	ERROR
		IF ERRNO = ERR_FILEOPEN THEN
			TPWrite "ERROR: Cannot open config.txt or log file";
		ELSE
			TPWrite "ERROR in TestGantryFloorCoordinates: " + NumToStr(ERRNO, 0);
		ENDIF
		Close configfile;
		Close debug_logfile;
		STOP;
	ENDPROC

	! ========================================
	! Test Gantry with Multiple R-axis Rotations
	! ========================================
	! Version: v1.8.7
	! Date: 2026-01-05
	! Purpose: Test Robot1 and Robot2 TCP positions at various R-axis angles
	! Features:
	!   - Config-based angle configuration (NUM_R_ANGLES, R_ANGLE_1~10)
	!   - Robot1 and Robot2 Floor TCP coordinate measurement
	!   - Automatic gantry position logging
	! Changes in v1.8.7:
	!   - Reduced header writes and summarized R_ANGLES for 41617 stability
	!   - Increased per-angle WaitTime to 0.2 for I/O stability
	! Changes in v1.8.5:
	!   - Log gantry Floor values using Floor conversion (X+9500, Y/Z inverted)
	! Changes in v1.8.4:
	!   - Chunked file logging with WaitTime 0.1 to reduce 41617
	! Changes in v1.8.1:
	!   - BUGFIX: Added UpdateRobot2BaseDynamicWobj() call (Line 1918)
	!   - Fixed Robot2 Floor TCP reporting [0,0,0]
	! Changes in v1.8.0:
	!   - Config-based R-axis angle reading from config.txt
	!   - Replaces hardcoded angles with NUM_R_ANGLES and R_ANGLE_1~10
	!   - Enhanced logging with gantry position details
	! Initial position: Robot1 and Robot2 at HOME
	! Gantry position: X=0, Y=0, Z=0 (fixed), R varies according to config
	! Output: /HOME/gantry_rotation_test.txt
	PROC TestGantryRotation()
		VAR jointtarget home_pos;
		VAR jointtarget test_pos;
		VAR robtarget rob1_floor;
		VAR robtarget rob2_floor;
		VAR iodev logfile;
		VAR iodev configfile;
		VAR num test_x;
		VAR num test_y;
		VAR num test_z;
		VAR num r_angles{10};
		VAR num num_r_angles;
		VAR num i;
		VAR string r_str;
		VAR string line;
		VAR string value_str;
		VAR string r_list;
		VAR string csv_line;
		VAR bool found_value;

		! Initialize
		test_x := 0;  ! Fixed at 0 for R-axis rotation test
		test_y := 0;
		test_z := 0;
		num_r_angles := 0;

		! Read config.txt for R angles
		TPWrite "Reading config.txt for R angles...";
		Open "HOME:/config.txt", configfile \Read;

		! Read NUM_R_ANGLES
		WHILE num_r_angles = 0 DO
			line := ReadStr(configfile \RemoveCR);
			IF StrFind(line, 1, "NUM_R_ANGLES=") = 1 THEN
				IF StrLen(line) >= 14 THEN
					value_str := StrPart(line, 14, StrLen(line) - 13);
					found_value := StrToVal(value_str, num_r_angles);
					TPWrite "NUM_R_ANGLES=" + NumToStr(num_r_angles, 0);
				ENDIF
			ENDIF
		ENDWHILE

		! Read R_ANGLE_1 to R_ANGLE_10
		FOR i FROM 1 TO num_r_angles DO
			WHILE TRUE DO
				line := ReadStr(configfile);
				IF StrFind(line, 1, "R_ANGLE_" + NumToStr(i,0) + "=") = 1 THEN
					value_str := StrPart(line, StrLen("R_ANGLE_" + NumToStr(i,0) + "=") + 1, StrLen(line) - StrLen("R_ANGLE_" + NumToStr(i,0) + "="));
					found_value := StrToVal(value_str, r_angles{i});
					TPWrite "R_ANGLE_" + NumToStr(i,0) + "=" + NumToStr(r_angles{i}, 1);
					GOTO next_angle;
				ENDIF
			ENDWHILE
			next_angle:
		ENDFOR

		Close configfile;

		! Build R angle list for header logging
		r_list := "";
		FOR i FROM 1 TO num_r_angles DO
			IF i = 1 THEN
				r_list := NumToStr(r_angles{i}, 1);
			ELSE
				r_list := r_list + "," + NumToStr(r_angles{i}, 1);
			ENDIF
		ENDFOR

		TPWrite "========================================";
		TPWrite "Starting Multiple R-axis Rotation Test";
		TPWrite "========================================";

		! Verify initial position
		TPWrite "Verifying robots at HOME position...";
		home_pos := CJointT();
		IF Abs(home_pos.extax.eax_a) > 10 OR Abs(home_pos.extax.eax_b) > 10 OR Abs(home_pos.extax.eax_c) > 10 OR Abs(home_pos.extax.eax_d) > 2 THEN
			TPWrite "WARNING: Gantry not at HOME!";
			TPWrite "Current: [" + NumToStr(home_pos.extax.eax_a,0) + ", " + NumToStr(home_pos.extax.eax_b,0) + ", " + NumToStr(home_pos.extax.eax_c,0) + ", " + NumToStr(home_pos.extax.eax_d,1) + "]";
			TPWrite "Please run SetRobot1InitialPosition first";
			RETURN;
		ENDIF

		! Open log file (reduced header writes)
		Open "HOME:/gantry_rotation_test.txt", logfile \Write;
		Write logfile, "Gantry R-axis Rotation Test (" + TASK1_VERSION + ")";
		Write logfile, "Date=" + CDate() + ", Time=" + CTime();
		Write logfile, "Gantry Phys=[" + NumToStr(test_x,0) + "," + NumToStr(test_y,0) + "," + NumToStr(test_z,0)
		              + "], Floor=[" + NumToStr(test_x + 9500,0) + "," + NumToStr(5300 - test_y,0) + "," + NumToStr(2100 - test_z,0) + "]";
		Write logfile, "R_ANGLES=" + r_list;
		Write logfile, "Floor: X+=right, Y+=up, Z+=up, R0:Y-axis, R1 Y+, R2 Y-";
		Write logfile, "R_DEG,GX,GY,GZ,R1X,R1Y,R1Z,R2X,R2Y,R2Z";
		WaitTime 0.3;

		! Test each R angle
		FOR i FROM 1 TO num_r_angles DO
			r_str := NumToStr(r_angles{i}, 1);
			TPWrite "----------------------------------------";
			TPWrite "Test " + NumToStr(i,0) + "/" + NumToStr(num_r_angles,0) + ": R = " + r_str + " degrees";
			TPWrite "----------------------------------------";

			! Move gantry to test position with current R angle
			test_pos := CJointT();
			test_pos.extax.eax_a := test_x;
			test_pos.extax.eax_b := test_y;
			test_pos.extax.eax_c := test_z;
			test_pos.extax.eax_d := r_angles{i};
			test_pos.extax.eax_f := test_x;  ! X2 = X1 (synchronized)
			MoveAbsJ test_pos, v100, fine, tool0;
			WaitTime 0.5;

			! Measure Floor positions
			UpdateRobot1FloorPosition;
			UpdateRobot2BaseDynamicWobj;  ! Update Robot2 base coordinate for TASK2
			! Note: robot2_floor_pos_t1 is updated by UpdateRobot2BaseDynamicWobj
			rob1_floor := robot1_floor_pos_t1;
			rob2_floor := robot2_floor_pos_t1;  ! Updated by TASK2

			! Write results to file (1-line CSV)
			csv_line := NumToStr(r_angles{i}, 1) + ","
			          + NumToStr(test_pos.extax.eax_a,0) + "," + NumToStr(test_pos.extax.eax_b,0) + "," + NumToStr(test_pos.extax.eax_c,0) + ","
			          + NumToStr(rob1_floor.trans.x, 2) + "," + NumToStr(rob1_floor.trans.y, 2) + "," + NumToStr(rob1_floor.trans.z, 2) + ","
			          + NumToStr(rob2_floor.trans.x, 2) + "," + NumToStr(rob2_floor.trans.y, 2) + "," + NumToStr(rob2_floor.trans.z, 2);
			Write logfile, csv_line;
			WaitTime 0.2; ! Keep this WaitTime for I/O stability
			! Display on teach pendant
			TPWrite "Robot1 Floor: [" + NumToStr(rob1_floor.trans.x,1) + ", " + NumToStr(rob1_floor.trans.y,1) + ", " + NumToStr(rob1_floor.trans.z,1) + "]";
			TPWrite "Robot2 Floor: [" + NumToStr(rob2_floor.trans.x,1) + ", " + NumToStr(rob2_floor.trans.y,1) + ", " + NumToStr(rob2_floor.trans.z,1) + "]";
		ENDFOR

		! Return to HOME
		TPWrite "Returning to HOME...";
		MoveAbsJ home_pos, v100, fine, tool0;

		Write logfile, "========================================";
		Write logfile, "Test completed - Returned to HOME";
		Write logfile, "========================================";
		Close logfile;

		TPWrite "========================================";
		TPWrite "R-axis Rotation Test Complete!";
		TPWrite "Results saved to gantry_rotation_test.txt";
		TPWrite "========================================";

	ERROR
		IF ERRNO = ERR_FILEOPEN THEN
			TPWrite "ERROR: Cannot open log file";
		ELSE
			TPWrite "ERROR in TestGantryRotation: " + NumToStr(ERRNO, 0);
		ENDIF
		Close logfile;
		STOP;
	ENDPROC

	! ========================================
	! Mode 2 - Gantry + TCP Offset Verification
	! ========================================
		! Version: v1.8.50
		! Date: 2026-01-08
		! Purpose: Verify TCP tracking with offsets while gantry moves in X/Y/Z/R
		! Config (config.txt):
		!   TEST_MODE=2
		!   TCP_OFFSET_R1_X/Y/Z (fallback: TCP_OFFSET_X/Y/Z)
		!   NUM_POS, POS_1_X/Y/Z/R ...
	! Output: /HOME/gantry_mode2_test.txt
		! Changes in v1.8.50:
		!   - Use hardcoded Mode2 defaults (config.txt ignored).
		! Changes in v1.8.49:
		!   - Remove CONTINUE usage in Mode2 parse loop for RAPID compatibility.
		! Changes in v1.8.48:
		!   - Rework Mode2 config parsing: single-pass ReadStr loop with guards.
		! Changes in v1.8.47:
		!   - TEMP: Bypass config.txt parsing and use default Mode2 offsets/positions.
		! Changes in v1.8.46:
		!   - Use ReadStr \RemoveCR in Mode2 parsing loops to avoid blocking on CRLF files.
		! Changes in v1.8.14:
		!   - Align gantry axis range checks with MOC.cfg (M1/M2/M3/M4 limits)

! ========================================
! Mode 2 - Gantry + TCP Offset Verification (v1.8.51)
! ========================================
! Version: v1.8.51
! Date: 2026-01-08
! Purpose: Verify TCP tracking with offsets using PERS variables
! No config.txt parsing - all settings from PERS variables
! Output: /HOME/gantry_mode2_test.txt
PROC TestGantryMode2()
	VAR jointtarget home_pos;
	VAR jointtarget test_pos;
	VAR robtarget offset_tcp;
	VAR robtarget rob1_floor;
	VAR robtarget rob2_floor;
	VAR iodev logfile;
	VAR num tcp_offset_x;
	VAR num tcp_offset_y;
	VAR num tcp_offset_z;
	VAR num num_pos;
	VAR num pos_x{10};
	VAR num pos_y{10};
	VAR num pos_z{10};
	VAR num pos_r{10};
	VAR num i;
	VAR string csv_line;
	VAR num floor_x;
	VAR num floor_y;
	VAR num floor_z;
	VAR num floor_r;
	VAR num phys_x;
	VAR num phys_y;
	VAR num phys_z;
	VAR num phys_r;
	VAR bool abort_test;
	VAR string mode2_log;
	VAR string tp_log;
	VAR iodev tp_logfile;
	VAR jointtarget current_gantry;
	VAR robjoint robot1_offset_joints;
	VAR num wait_count;

	abort_test := FALSE;
	mode2_log := "HOME:/gantry_mode2_test.txt";
	tp_log := "HOME:/tp_messages.txt";

	! v1.8.57: Reset sync flags at start (TASK2 must wait)
	mode2_config_ready := FALSE;
	mode2_r2_initial_offset_done := FALSE;

	Open mode2_log, logfile \Write;
	Open tp_log, tp_logfile \Write;
	Write tp_logfile, "TP Log (" + TASK1_VERSION + ") Date=" + CDate() + " Time=" + CTime();
	Write tp_logfile, "========================================";
	Write logfile, "Mode2 Test (" + TASK1_VERSION + ") Date=" + CDate() + " Time=" + CTime();
	Write logfile, "Enter TestGantryMode2";
	TPWrite "Mode2: Loading config from PERS variables";
	Write tp_logfile, "Mode2: Loading config from PERS variables";

	! DEBUG: Log ConfigModule PERS values BEFORE copy
	Write tp_logfile, "DEBUG: ConfigModule R2 BEFORE copy:";
	Write tp_logfile, "  MODE2_TCP_OFFSET_R2_X=" + NumToStr(MODE2_TCP_OFFSET_R2_X, 1);
	Write tp_logfile, "  MODE2_TCP_OFFSET_R2_Y=" + NumToStr(MODE2_TCP_OFFSET_R2_Y, 1);
	Write tp_logfile, "  MODE2_TCP_OFFSET_R2_Z=" + NumToStr(MODE2_TCP_OFFSET_R2_Z, 1);
	Write tp_logfile, "DEBUG: mode2_r2_offset BEFORE copy:";
	Write tp_logfile, "  mode2_r2_offset_y=" + NumToStr(mode2_r2_offset_y, 1);

	! Read configuration from PERS variables (no file I/O)
	tcp_offset_x := MODE2_TCP_OFFSET_R1_X;
	tcp_offset_y := MODE2_TCP_OFFSET_R1_Y;
	tcp_offset_z := MODE2_TCP_OFFSET_R1_Z;

	! Sync Robot2 offsets from ConfigModule (for TASK2)
	mode2_r2_offset_x := MODE2_TCP_OFFSET_R2_X;
	mode2_r2_offset_y := MODE2_TCP_OFFSET_R2_Y;
	mode2_r2_offset_z := MODE2_TCP_OFFSET_R2_Z;

	! v1.8.57: Set sync flag (TASK2 can now read values)
	mode2_config_ready := TRUE;
	Write tp_logfile, "SYNC: mode2_config_ready=TRUE (TASK2 can proceed)";

	! DEBUG: Log values AFTER copy
	Write tp_logfile, "DEBUG: mode2_r2_offset AFTER copy:";
	Write tp_logfile, "  mode2_r2_offset_y=" + NumToStr(mode2_r2_offset_y, 1);

	! Log Robot2 offsets
	Write logfile, "R2_OFFSET=" + NumToStr(mode2_r2_offset_x, 1) + ","
	              + NumToStr(mode2_r2_offset_y, 1) + ","
	              + NumToStr(mode2_r2_offset_z, 1);

	! Read test positions
	num_pos := MODE2_NUM_POS;
	FOR i FROM 1 TO 10 DO
		pos_x{i} := MODE2_POS_X{i};
		pos_y{i} := MODE2_POS_Y{i};
		pos_z{i} := MODE2_POS_Z{i};
		pos_r{i} := MODE2_POS_R{i};
	ENDFOR

	Write logfile, "Config loaded from PERS - NUM_POS=" + NumToStr(num_pos, 0);
	Write logfile, "TCP_OFFSET_R1=" + NumToStr(tcp_offset_x,1) + ","
	              + NumToStr(tcp_offset_y,1) + ","
	              + NumToStr(tcp_offset_z,1);
	Write logfile, "X,Y,Z,R,R1X,R1Y,R1Z,R2X,R2Y,R2Z";
	TPWrite "Mode2: Config loaded, NUM_POS=" + NumToStr(num_pos, 0);
	Write tp_logfile, "Mode2: Config loaded, NUM_POS=" + NumToStr(num_pos, 0);
	WaitTime 0.3;

	! Move Robot1 to offset in WobjGantry
	UpdateGantryWobj;
	home_pos := CJointT();
	offset_tcp := [[tcp_offset_x, tcp_offset_y, 1000 + tcp_offset_z], [0.5, -0.5, 0.5, 0.5], [0, 0, 0, 0], home_pos.extax];
	MoveJ offset_tcp, v100, fine, tool0\WObj:=WobjGantry;
	TPWrite "Mode2: Robot1 at offset TCP";
	Write tp_logfile, "Mode2: Robot1 at offset TCP";

	! Save Robot1 joint angles for use in loop (fixed joints = fixed TCP direction)
	current_gantry := CJointT();
	robot1_offset_joints := current_gantry.robax;
	Write tp_logfile, "Robot1 offset joints: saved";

	! v1.8.67: Wait for Robot2 initial offset before moving gantry
	TPWrite "Mode2: Waiting for Robot2 initial offset...";
	Write tp_logfile, "SYNC: Waiting for Robot2 initial offset...";
	wait_count := 0;
	WHILE NOT mode2_r2_initial_offset_done AND wait_count < 100 DO
		WaitTime 0.1;
		wait_count := wait_count + 1;
	ENDWHILE
	IF mode2_r2_initial_offset_done THEN
		Write tp_logfile, "SYNC: Robot2 initial offset done (waited " + NumToStr(wait_count, 0) + " cycles)";
		TPWrite "Mode2: Robot2 initial offset done";
	ELSE
		Write tp_logfile, "WARNING: Robot2 initial offset timeout!";
		TPWrite "Mode2: WARNING - Robot2 offset timeout!";
	ENDIF

	! Test each position
	FOR i FROM 1 TO num_pos DO
		! Calculate Floor coordinates (COMPLEX_POS format)
		floor_x := 9500 + pos_x{i};
		floor_y := 5300 + pos_y{i};
		floor_z := 2100 + pos_z{i};
		floor_r := pos_r{i};

		! Convert to physical gantry coordinates
		phys_x := floor_x - 9500;
		phys_y := 5300 - floor_y;
		phys_z := 2100 - floor_z;
		phys_r := 0 - floor_r;

		! Check gantry axis limits (MOC.cfg)
		! M1 [-9.51, 12.31], M2 [-0.05, 5.35], M3 [-0.05, 1.05], M4 [-100, 100] deg
		IF phys_x < -9510 OR phys_x > 12310 OR phys_y < -50 OR phys_y > 5350 OR phys_z < -50 OR phys_z > 1050 OR phys_r < -100 OR phys_r > 100 THEN
			Write logfile, "OUT_OF_RANGE idx=" + NumToStr(i,0)
			              + " floor=[" + NumToStr(floor_x,0) + "," + NumToStr(floor_y,0) + "," + NumToStr(floor_z,0) + "," + NumToStr(floor_r,1) + "]"
			              + " phys=[" + NumToStr(phys_x,0) + "," + NumToStr(phys_y,0) + "," + NumToStr(phys_z,0) + "," + NumToStr(phys_r,1) + "]";
			TPWrite "Mode2: Position " + NumToStr(i,0) + " out of range!";
			abort_test := TRUE;
			GOTO mode2_cleanup;
		ENDIF

		! Move gantry to test position (Robot1 joints fixed to offset position)
		test_pos := CJointT();
		test_pos.robax := robot1_offset_joints;  ! Keep Robot1 at offset position
		test_pos.extax.eax_a := phys_x;
		test_pos.extax.eax_b := phys_y;
		test_pos.extax.eax_c := phys_z;
		test_pos.extax.eax_d := phys_r;
		test_pos.extax.eax_f := test_pos.extax.eax_a;
		MoveAbsJ test_pos, v100, fine, tool0;
		TPWrite "Mode2: Gantry moved to position " + NumToStr(i,0) + "/" + NumToStr(num_pos,0);
		Write tp_logfile, "Mode2: Gantry moved to position " + NumToStr(i,0) + "/" + NumToStr(num_pos,0);

		! Update WobjGantry for new gantry position and rotation
		UpdateGantryWobj;

		! Read current gantry position AFTER move (fix for eax_e mismatch)
		current_gantry := CJointT();
		Write tp_logfile, "WobjGantry updated: [" + NumToStr(current_gantry.extax.eax_a,0) + ", "
		                  + NumToStr(current_gantry.extax.eax_b,0) + ", "
		                  + NumToStr(current_gantry.extax.eax_c,0) + ", R="
		                  + NumToStr(current_gantry.extax.eax_d,1) + "]";
		Write tp_logfile, "current_gantry.extax: [" + NumToStr(current_gantry.extax.eax_a,1) + ", "
		                  + NumToStr(current_gantry.extax.eax_b,1) + ", "
		                  + NumToStr(current_gantry.extax.eax_c,1) + ", "
		                  + NumToStr(current_gantry.extax.eax_d,1) + ", "
		                  + NumToStr(current_gantry.extax.eax_e,1) + ", "
		                  + NumToStr(current_gantry.extax.eax_f,1) + "]";

		! Robot1 already at offset position (joints fixed in MoveAbsJ)
		Write tp_logfile, "Robot1 maintaining offset joints (pos " + NumToStr(i,0) + ")";

		! v1.8.63: Trigger Robot2 to reposition at current R angle
		mode2_r2_reposition_done := FALSE;
		mode2_r2_reposition_trigger := TRUE;
		Write tp_logfile, "SYNC: Waiting for Robot2 reposition...";
		wait_count := 0;
		WHILE NOT mode2_r2_reposition_done AND wait_count < 100 DO
			WaitTime 0.1;
			wait_count := wait_count + 1;
		ENDWHILE
		mode2_r2_reposition_trigger := FALSE;
		IF mode2_r2_reposition_done THEN
			Write tp_logfile, "SYNC: Robot2 repositioned (waited " + NumToStr(wait_count, 0) + " cycles)";
		ELSE
			Write tp_logfile, "SYNC: WARNING - Robot2 reposition timeout!";
		ENDIF
		WaitTime 0.3;

		! Measure Robot1 and Robot2 TCP positions
		UpdateRobot1FloorPosition;
		UpdateRobot2BaseDynamicWobj;
		rob1_floor := robot1_floor_pos_t1;
		rob2_floor := robot2_floor_pos_t1;

		! v1.8.60 DEBUG: Detailed position analysis
		Write tp_logfile, "========== v1.8.60 DETAILED DEBUG ==========";
		Write tp_logfile, "--- Gantry Position ---";
		Write tp_logfile, "  Gantry Floor: [" + NumToStr(floor_x, 0) + ", " + NumToStr(floor_y, 0) + ", " + NumToStr(floor_z, 0) + "]";
		Write tp_logfile, "  Gantry Local (extax): [" + NumToStr(phys_x, 0) + ", " + NumToStr(phys_y, 0) + ", " + NumToStr(phys_z, 0) + ", R=" + NumToStr(phys_r, 1) + "]";
		Write tp_logfile, "  R-center Floor: [" + NumToStr(floor_x, 0) + ", " + NumToStr(floor_y, 0) + ", " + NumToStr(floor_z, 0) + "]";
		Write tp_logfile, "";
		Write tp_logfile, "--- Robot1 (wobj0 at R-center, gantry-configured) ---";
		Write tp_logfile, "  Robot1 Base Floor = R-center: [" + NumToStr(floor_x, 0) + ", " + NumToStr(floor_y, 0) + ", " + NumToStr(floor_z, 0) + "]";
		Write tp_logfile, "  Robot1 offset_tcp in WobjGantry: [" + NumToStr(tcp_offset_x, 1) + ", " + NumToStr(tcp_offset_y, 1) + ", " + NumToStr(1000 + tcp_offset_z, 1) + "]";
		Write tp_logfile, "  Robot1 TCP Floor (measured): [" + NumToStr(rob1_floor.trans.x, 2) + ", " + NumToStr(rob1_floor.trans.y, 2) + ", " + NumToStr(rob1_floor.trans.z, 2) + "]";
		Write tp_logfile, "  Robot1 TCP offset from R-center: [" + NumToStr(rob1_floor.trans.x - floor_x, 2) + ", " + NumToStr(rob1_floor.trans.y - floor_y, 2) + ", " + NumToStr(rob1_floor.trans.z - floor_z, 2) + "]";
		Write tp_logfile, "";
		Write tp_logfile, "--- Robot2 (wobj0 at Robot2 base, NOT gantry-configured) ---";
		Write tp_logfile, "  Robot2 Base Floor: [" + NumToStr(debug_r2_base_floor_x, 2) + ", " + NumToStr(rob2_floor.trans.y - (debug_r2_wobj0_y * Cos(current_gantry.extax.eax_d)), 2) + "]";
		Write tp_logfile, "  Robot2 offset_tcp in WobjGantry_Rob2: [0, " + NumToStr(488 + mode2_r2_offset_y, 1) + ", -1000]";
		Write tp_logfile, "  Robot2 wobj0 (TCP from base): [" + NumToStr(debug_r2_wobj0_x, 2) + ", " + NumToStr(debug_r2_wobj0_y, 2) + "]";
		Write tp_logfile, "  Robot2 TCP Floor (measured): [" + NumToStr(rob2_floor.trans.x, 2) + ", " + NumToStr(rob2_floor.trans.y, 2) + ", " + NumToStr(rob2_floor.trans.z, 2) + "]";
		Write tp_logfile, "  Robot2 TCP offset from R-center: [" + NumToStr(rob2_floor.trans.x - floor_x, 2) + ", " + NumToStr(rob2_floor.trans.y - floor_y, 2) + ", " + NumToStr(rob2_floor.trans.z - floor_z, 2) + "]";
		Write tp_logfile, "";
		Write tp_logfile, "--- Comparison ---";
		Write tp_logfile, "  3D Distance: " + NumToStr(Sqrt(Pow(rob1_floor.trans.x - rob2_floor.trans.x, 2) + Pow(rob1_floor.trans.y - rob2_floor.trans.y, 2) + Pow(rob1_floor.trans.z - rob2_floor.trans.z, 2)), 2) + " mm";
		Write tp_logfile, "  Expected (at R=0): 200.00 mm";
		Write tp_logfile, "=========================================";

		! v1.8.61 DEBUG: Log X coordinate analysis
		Write tp_logfile, "DEBUG X Analysis:";
		Write tp_logfile, "  Gantry X (R-center): " + NumToStr(phys_x + 9500, 1);
		Write tp_logfile, "  R angle (extax.eax_d): " + NumToStr(current_gantry.extax.eax_d, 1);
		Write tp_logfile, "  sin(R): " + NumToStr(Sin(current_gantry.extax.eax_d), 4);
		Write tp_logfile, "  Robot2 wobj0: [" + NumToStr(debug_r2_wobj0_x, 1) + ", " + NumToStr(debug_r2_wobj0_y, 1) + "]";
		Write tp_logfile, "  Robot2 base_floor_x: " + NumToStr(debug_r2_base_floor_x, 1);
		Write tp_logfile, "  Robot2 floor_x_offset: " + NumToStr(debug_r2_floor_x_offset, 1);
		Write tp_logfile, "  Robot2 X = base + offset: " + NumToStr(debug_r2_base_floor_x, 1) + " + " + NumToStr(debug_r2_floor_x_offset, 1) + " = " + NumToStr(rob2_floor.trans.x, 1);
		Write tp_logfile, "  Robot1 X: " + NumToStr(rob1_floor.trans.x, 2) + " (offset from gantry: " + NumToStr(rob1_floor.trans.x - (phys_x + 9500), 2) + ")";
		Write tp_logfile, "  Robot2 X: " + NumToStr(rob2_floor.trans.x, 2) + " (offset from gantry: " + NumToStr(rob2_floor.trans.x - (phys_x + 9500), 2) + ")";
		Write tp_logfile, "  Expected R2 X offset: +" + NumToStr(100 * Sin(current_gantry.extax.eax_d), 2);
		Write tp_logfile, "  Delta X (R1-R2): " + NumToStr(rob1_floor.trans.x - rob2_floor.trans.x, 2);

		! v1.8.61 DEBUG: Log Y coordinate analysis
		Write tp_logfile, "DEBUG Y Analysis:";
		Write tp_logfile, "  Gantry Y (R-center): " + NumToStr(5300 - phys_y, 1);
		Write tp_logfile, "  cos(R): " + NumToStr(Cos(current_gantry.extax.eax_d), 4);
		Write tp_logfile, "  Robot2 base_floor_y: " + NumToStr(debug_r2_base_floor_y, 1);
		Write tp_logfile, "  Robot2 floor_y_offset: " + NumToStr(debug_r2_floor_y_offset, 1);
		Write tp_logfile, "  Robot2 Y = base + offset: " + NumToStr(debug_r2_base_floor_y, 1) + " + " + NumToStr(debug_r2_floor_y_offset, 1) + " = " + NumToStr(rob2_floor.trans.y, 1);
		Write tp_logfile, "  Robot1 Y: " + NumToStr(rob1_floor.trans.y, 2) + " (offset from gantry: " + NumToStr(rob1_floor.trans.y - (5300 - phys_y), 2) + ")";
		Write tp_logfile, "  Robot2 Y: " + NumToStr(rob2_floor.trans.y, 2) + " (offset from gantry: " + NumToStr(rob2_floor.trans.y - (5300 - phys_y), 2) + ")";
		Write tp_logfile, "  Expected R1 Y offset: +" + NumToStr(100 * Cos(current_gantry.extax.eax_d), 2);
		Write tp_logfile, "  Expected R2 Y offset: -" + NumToStr(100 * Cos(current_gantry.extax.eax_d), 2);
		Write tp_logfile, "  Delta Y (R1-R2): " + NumToStr(rob1_floor.trans.y - rob2_floor.trans.y, 2);
		Write tp_logfile, "  Expected Delta Y: " + NumToStr(200 * Cos(current_gantry.extax.eax_d), 2);

		Write tp_logfile, "Robot1 Floor: [" + NumToStr(rob1_floor.trans.x,2) + ", " + NumToStr(rob1_floor.trans.y,2) + ", " + NumToStr(rob1_floor.trans.z,2) + "]";
		Write tp_logfile, "Robot2 Floor: [" + NumToStr(rob2_floor.trans.x,2) + ", " + NumToStr(rob2_floor.trans.y,2) + ", " + NumToStr(rob2_floor.trans.z,2) + "]";
		Write tp_logfile, "----------------------------------------";

		! Log result
		csv_line := NumToStr(floor_x,0) + "," + NumToStr(floor_y,0) + "," + NumToStr(floor_z,0) + "," + NumToStr(floor_r,1) + ","
		          + NumToStr(rob1_floor.trans.x, 2) + "," + NumToStr(rob1_floor.trans.y, 2) + "," + NumToStr(rob1_floor.trans.z, 2) + ","
		          + NumToStr(rob2_floor.trans.x, 2) + "," + NumToStr(rob2_floor.trans.y, 2) + "," + NumToStr(rob2_floor.trans.z, 2);
		Write logfile, csv_line;
		WaitTime 0.2;
	ENDFOR

mode2_cleanup:
	! Always return gantry to HOME
	TPWrite "Mode2: Returning to HOME";
	Write tp_logfile, "Mode2: Returning to HOME";
	home_pos := CJointT();
	home_pos.extax.eax_a := 0;
	home_pos.extax.eax_b := 0;
	home_pos.extax.eax_c := 0;
	home_pos.extax.eax_d := 0;
	home_pos.extax.eax_f := 0;
	MoveAbsJ home_pos, v100, fine, tool0;

	TPWrite "Mode2: Test complete!";
	Write tp_logfile, "Mode2: Test complete!";
	Write tp_logfile, "========================================";

	! v1.8.63: Signal TASK2 to exit reposition monitor loop
	mode2_config_ready := FALSE;

	Close logfile;
	Close tp_logfile;
	IF abort_test = TRUE THEN
		TPWrite "Mode2: Test aborted (out of range)";
		STOP;
	ENDIF

ERROR
	Write logfile, "ERROR in TestGantryMode2: " + NumToStr(ERRNO, 0);
	Write tp_logfile, "ERROR in TestGantryMode2: " + NumToStr(ERRNO, 0);
	Close logfile;
	Close tp_logfile;
	TPWrite "ERROR in TestGantryMode2: " + NumToStr(ERRNO, 0);
	STOP;
ENDPROC

! ========================================
! TestInitNonHome - Automated Non-HOME Init Verification (v1.9.50)
! ========================================
! Purpose: Verify SetRobot1InitialPosition works correctly when gantry
!          starts at non-HOME positions (4 scenarios: HOME, R=30, XYZ, XYZ+R=30)
! Output:  HOME:/test_init_nonhome.txt
PROC TestInitNonHome()
    VAR iodev test_logfile;
    VAR jointtarget gantry_pos;
    VAR robtarget tcp_gantry;
    VAR robtarget tcp_floor;
    VAR num test_floor_x{4};
    VAR num test_floor_y{4};
    VAR num test_floor_z{4};
    VAR num test_floor_r{4};
    VAR string test_name{4};
    VAR num pass_count;
    VAR num err_x;
    VAR num err_y;
    VAR num err_z;
    VAR bool scenario_pass;
    VAR string result_str;
    VAR jointtarget jt_after;

    ! Define 4 test scenarios (Floor coordinates)
    test_name{1} := "A:HOME";        test_floor_x{1}:=9500; test_floor_y{1}:=5300; test_floor_z{1}:=2100; test_floor_r{1}:=0;
    test_name{2} := "B:R=30";        test_floor_x{2}:=9500; test_floor_y{2}:=5300; test_floor_z{2}:=2100; test_floor_r{2}:=30;
    test_name{3} := "C:XYZ";         test_floor_x{3}:=8500; test_floor_y{3}:=5000; test_floor_z{3}:=1900; test_floor_r{3}:=0;
    test_name{4} := "D:XYZ+R=30";    test_floor_x{4}:=8500; test_floor_y{4}:=5000; test_floor_z{4}:=1900; test_floor_r{4}:=30;

    Open "HOME:/test_init_nonhome.txt", test_logfile \Write;
    Write test_logfile, "=== TestInitNonHome (" + TASK1_VERSION + ") ===";
    Write test_logfile, "Date=" + CDate() + " Time=" + CTime();
    Write test_logfile, "";
    WaitTime 0.3;

    pass_count := 0;

    FOR i FROM 1 TO 4 DO
        TPWrite "--- Scenario " + test_name{i} + " ---";
        Write test_logfile, "========================================";
        Write test_logfile, "Scenario " + test_name{i};
        Write test_logfile, "  Floor: X=" + NumToStr(test_floor_x{i},0) + " Y=" + NumToStr(test_floor_y{i},0) + " Z=" + NumToStr(test_floor_z{i},0) + " R=" + NumToStr(test_floor_r{i},0);

        ! Convert Floor -> Physical and move gantry
        gantry_pos := CJointT();
        gantry_pos.extax.eax_a := test_floor_x{i} - 9500;
        gantry_pos.extax.eax_b := 5300 - test_floor_y{i};
        gantry_pos.extax.eax_c := 2100 - test_floor_z{i};
        gantry_pos.extax.eax_d := 0 - test_floor_r{i};
        gantry_pos.extax.eax_f := test_floor_x{i} - 9500;  ! X2=X1
        MoveAbsJ gantry_pos, v200, fine, tool0;
        WaitTime 0.5;

        Write test_logfile, "  Phys: eax_a=" + NumToStr(gantry_pos.extax.eax_a,1) + " b=" + NumToStr(gantry_pos.extax.eax_b,1) + " c=" + NumToStr(gantry_pos.extax.eax_c,1) + " d=" + NumToStr(gantry_pos.extax.eax_d,1);
        Write test_logfile, "  Calling SetRobot1InitialPosition...";
        WaitTime 0.2;

        ! Call init (this moves gantry back to HOME internally at Step 3)
        SetRobot1InitialPosition;

        ! After init: gantry is at HOME, robot TCP should be correct
        ! Read TCP in WobjGantry (should be near [0, 0, 1000])
        UpdateGantryWobj;
        tcp_gantry := CRobT(\Tool:=tWeld1\WObj:=WobjGantry);
        ! Read TCP in WobjFloor (should be consistent across all scenarios)
        tcp_floor := CRobT(\Tool:=tWeld1\WObj:=WobjFloor);

        err_x := Abs(tcp_gantry.trans.x - 0);
        err_y := Abs(tcp_gantry.trans.y - 0);
        err_z := Abs(tcp_gantry.trans.z - 1000);
        scenario_pass := (err_x < 1) AND (err_y < 1) AND (err_z < 1);

        IF scenario_pass THEN
            pass_count := pass_count + 1;
            result_str := "PASS";
        ELSE
            result_str := "FAIL";
        ENDIF

        ! Read joint angles after init
        jt_after := CJointT();

        Write test_logfile, "  Result: " + result_str;
        Write test_logfile, "  TCP_Gantry: [" + NumToStr(tcp_gantry.trans.x,3) + ", " + NumToStr(tcp_gantry.trans.y,3) + ", " + NumToStr(tcp_gantry.trans.z,3) + "]";
        Write test_logfile, "  TCP_Gantry orient: [" + NumToStr(tcp_gantry.rot.q1,5) + ", " + NumToStr(tcp_gantry.rot.q2,5) + ", " + NumToStr(tcp_gantry.rot.q3,5) + ", " + NumToStr(tcp_gantry.rot.q4,5) + "]";
        Write test_logfile, "  TCP_Floor: [" + NumToStr(tcp_floor.trans.x,1) + ", " + NumToStr(tcp_floor.trans.y,1) + ", " + NumToStr(tcp_floor.trans.z,1) + "]";
        Write test_logfile, "  Joints: [" + NumToStr(jt_after.robax.rax_1,2) + ", " + NumToStr(jt_after.robax.rax_2,2) + ", " + NumToStr(jt_after.robax.rax_3,2) + ", " + NumToStr(jt_after.robax.rax_4,2) + ", " + NumToStr(jt_after.robax.rax_5,2) + ", " + NumToStr(jt_after.robax.rax_6,2) + "]";
        Write test_logfile, "  Error: dX=" + NumToStr(err_x,3) + " dY=" + NumToStr(err_y,3) + " dZ=" + NumToStr(err_z,3);
        Write test_logfile, "";
        WaitTime 0.3;

        TPWrite test_name{i} + ": " + result_str + " dX=" + NumToStr(err_x,2) + " dY=" + NumToStr(err_y,2);
    ENDFOR

    ! Summary
    Write test_logfile, "========================================";
    Write test_logfile, "SUMMARY: " + NumToStr(pass_count,0) + "/4 PASSED";
    Write test_logfile, "========================================";
    Close test_logfile;

    TPWrite "TestInitNonHome: " + NumToStr(pass_count,0) + "/4 passed";
    TPWrite "Log: HOME:/test_init_nonhome.txt";
ENDPROC

! ========================================
! Test Menu System (v1.9.2)
! ========================================
! Purpose: TP-based menu for test selection
! Options: Mode2 Test, Weld Sequence, View Results, Exit

! ----------------------------------------
! Main Test Menu
! ----------------------------------------
! Displays menu on TP and executes selected test
! Loop until user selects Exit
PROC TestMenu()
	VAR num menu_sel;
	VAR bool menu_loop;

	menu_loop := TRUE;

	WHILE menu_loop DO
		! Display menu
		TPErase;
		TPWrite "========================================";
		TPWrite "  S25016 SpGantry Test Menu (v2.8.0)";
		TPWrite "========================================";
		TPWrite "";
		TPWrite "  1. Sync X1/X2 (Check + Auto-fix)";
		TPWrite "  2. Edge to Weld (CALC ONLY, no move)";
		TPWrite "  3. Edge to Weld (with gantry move)";
		TPWrite "  4. Test Gantry Floor Coordinates";
		TPWrite "  5. Execute Weld Sequence";
		TPWrite "  6. View Config";
		TPWrite "  7. View Results";
		TPWrite "  8. Multi-Angle Test (0/45/90/-45 deg)";
		TPWrite "  9. Edge to Weld + Robot1 Move";
		TPWrite " 10. Multi-Position Test (5 locations)";
		TPWrite " 11. Full Weld Seq (Gantry+R1+R2 sync)";
		TPWrite " 12. Init Non-HOME Test (4 scenarios)";
		TPWrite " 13. Guard Test (#8 TC T1~T5)";
		TPWrite " 14. Swap Scenarios (A~E auto)";
		TPWrite " 15. [Hybrid] DefineWeldLine->Gantry Stage1";
		TPWrite "  0. Exit";
		TPWrite "";
		TPWrite "----------------------------------------";

		! Numeric selection
		TPReadNum menu_sel, "Select (0-15): ";

		TEST menu_sel
		CASE 1:
			TPErase;
			TPWrite "[Menu] Checking Linked Motor Sync...";
			CheckLinkedMotorSync;
			TPWrite "";
			TPWrite "Press any key to continue...";
			TPReadFK menu_sel, "Continue?", "OK", "", "", "", "";

		CASE 2:
			TPErase;
			TPWrite "[Menu] Edge to Weld CALC ONLY...";
			TestEdgeToWeldCalcOnly;
			TPWrite "";
			TPWrite "Press any key to continue...";
			TPReadFK menu_sel, "Continue?", "OK", "", "", "", "";

		CASE 3:
			TPErase;
			TPWrite "[Menu] Edge to Weld with Movement...";
			TestEdgeToWeld;
			TPWrite "";
			TPWrite "Press any key to continue...";
			TPReadFK menu_sel, "Continue?", "OK", "", "", "", "";

		CASE 4:
			TPErase;
			TPWrite "[Menu] Starting Floor Coordinate Test...";
			TestGantryFloorCoordinates;
			TPWrite "";
			TPWrite "Press any key to continue...";
			TPReadFK menu_sel, "Continue?", "OK", "", "", "", "";

		CASE 5:
			TPErase;
			TPWrite "[Menu] Starting Weld Sequence...";
			ExecuteWeldSequence;
			TPWrite "";
			TPWrite "Press any key to continue...";
			TPReadFK menu_sel, "Continue?", "OK", "", "", "", "";

		CASE 6:
			TPErase;
			ViewCurrentConfig;
			TPWrite "";
			TPWrite "Press any key to continue...";
			TPReadFK menu_sel, "Continue?", "OK", "", "", "", "";

		CASE 7:
			TPErase;
			ViewLastResults;
			TPWrite "";
			TPWrite "Press any key to continue...";
			TPReadFK menu_sel, "Continue?", "OK", "", "", "", "";

		CASE 8:
			TPErase;
			TPWrite "[Menu] Starting Multi-Angle Test...";
			TestMultiAngle;
			TPWrite "";
			TPWrite "Press any key to continue...";
			TPReadFK menu_sel, "Continue?", "OK", "", "", "", "";

		CASE 9:
			TPErase;
			TPWrite "[Menu] Edge to Weld + Robot Move...";
			TestEdgeToWeldWithRobot;
			TPWrite "";
			TPWrite "Press any key to continue...";
			TPReadFK menu_sel, "Continue?", "OK", "", "", "", "";

		CASE 10:
			TPErase;
			TPWrite "[Menu] Starting Multi-Position Test...";
			TestMultiPosition;
			TPWrite "";
			TPWrite "Press any key to continue...";
			TPReadFK menu_sel, "Continue?", "OK", "", "", "", "";

		CASE 11:
			TPErase;
			TPWrite "[Menu] Full Weld Sequence (Gantry+R1+R2)...";
			TPWrite "NOTE: TASK2 must be in Weld mode";
			TestFullWeldSequence;
			TPWrite "";
			TPWrite "Press any key to continue...";
			TPReadFK menu_sel, "Continue?", "OK", "", "", "", "";

		CASE 12:
			TPErase;
			TPWrite "[Menu] Init Non-HOME Test (v1.9.49 verification)...";
			TestInitNonHome;
			TPWrite "";
			TPWrite "Press any key to continue...";
			TPReadFK menu_sel, "Continue?", "OK", "", "", "", "";

		CASE 13:
			TPErase;
			TPWrite "[Menu] Guard Verification (#8 TC T1~T5)...";
			TestGuardVerification;
			TPWrite "";
			TPWrite "Press any key to continue...";
			TPReadFK menu_sel, "Continue?", "OK", "", "", "", "";

		CASE 14:
			TPErase;
			TPWrite "[Menu] Swap Scenarios (A~E auto)...";
			TestSwapScenarios;
			TPWrite "";
			TPWrite "Press any key to continue...";
			TPReadFK menu_sel, "Continue?", "OK", "", "", "", "";

		CASE 15:
			TPErase;
			TPWrite "[Menu] Hybrid: DefineWeldLine->Gantry Stage1...";
			TestPlanAB_Stage1;
			TPWrite "";
			TPWrite "Press any key to continue...";
			TPReadFK menu_sel, "Continue?", "OK", "", "", "", "";

		CASE 0:
			TPErase;
			TPWrite "[Menu] Exiting Test Menu...";
			menu_loop := FALSE;

		DEFAULT:
			TPWrite "[Menu] Invalid selection (0-14)";
			WaitTime 1;
		ENDTEST
	ENDWHILE

	TPWrite "========================================";
	TPWrite "Test Menu closed. Returning to main...";
	TPWrite "========================================";
ENDPROC

! ----------------------------------------
! View Last Test Results
! ----------------------------------------
! Displays summary of last Mode2 test results
PROC ViewLastResults()
	VAR iodev resultfile;
	VAR string line;
	VAR num line_count;
	VAR bool file_ok;

	TPWrite "========================================";
	TPWrite "  Last Mode2 Test Results";
	TPWrite "========================================";
	TPWrite "";

	file_ok := TRUE;
	Open "HOME:/gantry_mode2_test.txt", resultfile \Read;

	! Read and display first 15 lines
	line_count := 0;
	WHILE file_ok AND line_count < 15 DO
		line := ReadStr(resultfile \Delim:="\0a");
		IF StrLen(line) > 0 THEN
			TPWrite line;
			line_count := line_count + 1;
		ENDIF
	ENDWHILE

	Close resultfile;

	TPWrite "";
	TPWrite "----------------------------------------";
	TPWrite "Full log: HOME:/gantry_mode2_test.txt";
	TPWrite "TP log: HOME:/tp_messages.txt";

ERROR
	IF ERRNO = ERR_FILEOPEN THEN
		TPWrite "ERROR: Result file not found";
		TPWrite "Run Mode2 test first!";
		file_ok := FALSE;
		TRYNEXT;
	ELSE
		! End of file or other read error
		Close resultfile;
		file_ok := FALSE;
		TRYNEXT;
	ENDIF
ENDPROC

! ----------------------------------------
! View Current Configuration
! ----------------------------------------
! Displays current Mode2 and Weld configuration
PROC ViewCurrentConfig()
	TPWrite "========================================";
	TPWrite "  Current Configuration (v1.9.2)";
	TPWrite "========================================";
	TPWrite "";

	TPWrite "--- Mode2 TCP Offsets ---";
	TPWrite "R1 Offset: [" + NumToStr(MODE2_TCP_OFFSET_R1_X, 1) + ", "
	                       + NumToStr(MODE2_TCP_OFFSET_R1_Y, 1) + ", "
	                       + NumToStr(MODE2_TCP_OFFSET_R1_Z, 1) + "]";
	TPWrite "R2 Offset: [" + NumToStr(MODE2_TCP_OFFSET_R2_X, 1) + ", "
	                       + NumToStr(MODE2_TCP_OFFSET_R2_Y, 1) + ", "
	                       + NumToStr(MODE2_TCP_OFFSET_R2_Z, 1) + "]";
	TPWrite "Num Positions: " + NumToStr(MODE2_NUM_POS, 0);
	TPWrite "";

	TPWrite "--- Weld Sequence ---";
	TPWrite "R1 Start: [" + NumToStr(WELD_R1_START_X, 0) + ", "
	                      + NumToStr(WELD_R1_START_Y, 0) + ", "
	                      + NumToStr(WELD_R1_START_Z, 0) + "]";
	TPWrite "R1 End: [" + NumToStr(WELD_R1_END_X, 0) + ", "
	                    + NumToStr(WELD_R1_END_Y, 0) + ", "
	                    + NumToStr(WELD_R1_END_Z, 0) + "]";
	TPWrite "R2 Start: [" + NumToStr(WELD_R2_START_X, 0) + ", "
	                      + NumToStr(WELD_R2_START_Y, 0) + ", "
	                      + NumToStr(WELD_R2_START_Z, 0) + "]";
	TPWrite "R2 End: [" + NumToStr(WELD_R2_END_X, 0) + ", "
	                    + NumToStr(WELD_R2_END_Y, 0) + ", "
	                    + NumToStr(WELD_R2_END_Z, 0) + "]";
	TPWrite "";

	TPWrite "--- Weld Robot Positions (WObj) ---";
	TPWrite "R1 WObj: [" + NumToStr(WELD_R1_WObj_X, 0) + ", "
	                     + NumToStr(WELD_R1_WObj_Y, 0) + ", "
	                     + NumToStr(WELD_R1_WObj_Z, 0) + "]";
	TPWrite "R2 WObj: [" + NumToStr(WELD_R2_WObj_X, 0) + ", "
	                     + NumToStr(WELD_R2_WObj_Y, 0) + ", "
	                     + NumToStr(WELD_R2_WObj_Z, 0) + "]";
	TPWrite "TCP Z Offset: " + NumToStr(WELD_R1_TCP_Z_OFFSET, 0) + " mm";
	TPWrite "Weld Speed: " + NumToStr(WELD_SPEED, 0) + " mm/s";
ENDPROC

! ========================================
! Weld Sequence Procedures (v1.9.0)
! ========================================
! Purpose: Execute welding sequence with calculated gantry position
! Input: Weld lines from ConfigModule PERS variables
! Output: Gantry moves along center line while robots maintain weld posture

! ----------------------------------------
! Calculate Center Line from Two Weld Lines
! ----------------------------------------
! Calculates center point between Robot1 and Robot2 weld lines
! Sets module variables: weld_center_start, weld_center_end, weld_center_angle, weld_length
PROC CalcCenterLine()
	VAR num dx;
	VAR num dy;
	VAR num dz;

	TPWrite "[WELD] Calculating center line...";

	! Calculate center start point (average of R1 and R2 start)
	weld_center_start.x := (WELD_R1_START_X + WELD_R2_START_X) / 2;
	weld_center_start.y := (WELD_R1_START_Y + WELD_R2_START_Y) / 2;
	weld_center_start.z := (WELD_R1_START_Z + WELD_R2_START_Z) / 2;

	! Calculate center end point (average of R1 and R2 end)
	weld_center_end.x := (WELD_R1_END_X + WELD_R2_END_X) / 2;
	weld_center_end.y := (WELD_R1_END_Y + WELD_R2_END_Y) / 2;
	weld_center_end.z := (WELD_R1_END_Z + WELD_R2_END_Z) / 2;

	! Calculate weld direction vector
	dx := weld_center_end.x - weld_center_start.x;
	dy := weld_center_end.y - weld_center_start.y;
	dz := weld_center_end.z - weld_center_start.z;

	! Calculate weld length
	weld_length := Sqrt(dx*dx + dy*dy + dz*dz);

	! Calculate R-axis angle (Floor X+ = R=0deg)
	! atan2(dy, dx) gives angle from X-axis
	weld_center_angle := ATan2(dy, dx);

	TPWrite "[WELD] Center Start: [" + NumToStr(weld_center_start.x, 1) + ", "
	                                  + NumToStr(weld_center_start.y, 1) + ", "
	                                  + NumToStr(weld_center_start.z, 1) + "]";
	TPWrite "[WELD] Center End: [" + NumToStr(weld_center_end.x, 1) + ", "
	                                + NumToStr(weld_center_end.y, 1) + ", "
	                                + NumToStr(weld_center_end.z, 1) + "]";
	TPWrite "[WELD] R-angle: " + NumToStr(weld_center_angle, 2) + " deg";
	TPWrite "[WELD] Weld length: " + NumToStr(weld_length, 1) + " mm";
ENDPROC

! ----------------------------------------
! Calculate Gantry Position from Floor Coordinates
! ----------------------------------------
! Converts Floor TCP coordinates to Physical gantry coordinates
! Accounts for robot TCP offset from R-center
! Gantry_Z = 2100 - Floor_Z - TCP_Z_OFFSET
FUNC pos CalcGantryFromFloor(pos floor_pos)
	VAR pos gantry_pos;

	! v1.9.58: Use Robot1 TCP offset only (TASK1 controls Robot1)
	! Robot1=1000mm (downward), Robot2=-1000mm (inverted) - averaging cancels out
	! Gantry Z positions R-center so Robot1 TCP reaches Floor Z target

	! Floor -> Physical conversion
	! gantry_x = floor_x - 9500
	! gantry_y = 5300 - floor_y
	! gantry_z = 2100 - floor_z - R1_tcp_offset
	gantry_pos.x := floor_pos.x - 9500;
	gantry_pos.y := 5300 - floor_pos.y;
	gantry_pos.z := 2100 - floor_pos.z - WELD_R1_TCP_Z_OFFSET;

	TPWrite "[WELD] Floor->Gantry: R1 TCP offset=" + NumToStr(WELD_R1_TCP_Z_OFFSET, 0) + "mm";
	TPWrite "[WELD] Gantry Z = 2100 - " + NumToStr(floor_pos.z, 0) + " - " + NumToStr(WELD_R1_TCP_Z_OFFSET, 0) + " = " + NumToStr(gantry_pos.z, 0);

	RETURN gantry_pos;
ENDFUNC

! ----------------------------------------
! Create Weld WObj from Weld Line
! ----------------------------------------
! Creates a work object where X-axis is weld direction, Z-axis is Floor Z (down)
! Parameters:
!   weld_start: Weld line start point (Floor coordinates)
!   weld_end: Weld line end point (Floor coordinates)
!   wobj: Output work object to update
PROC CreateWeldWobj(pos weld_start, pos weld_end, INOUT wobjdata wobj)
	VAR num dx;
	VAR num dy;
	VAR num len_xy;
	VAR num angle_deg;
	VAR num cos_half;
	VAR num sin_half;

	! Calculate weld direction in XY plane
	dx := weld_end.x - weld_start.x;
	dy := weld_end.y - weld_start.y;
	len_xy := Sqrt(dx*dx + dy*dy);

	! Calculate angle from X-axis (Floor X+ = 0 deg)
	! WObj X+ will align with weld direction
	angle_deg := ATan2(dy, dx);

	! Create quaternion for Z-axis rotation
	! Rotation around Z-axis by angle_deg
	! q = [cos(a/2), 0, 0, sin(a/2)]
	cos_half := Cos(angle_deg / 2);
	sin_half := Sin(angle_deg / 2);

	! Set WObj properties
	wobj.robhold := FALSE;
	wobj.ufprog := TRUE;
	wobj.ufmec := "";

	! Set uframe (user frame): origin at weld start, rotated around Z
	! WObj X = weld direction, Y = perpendicular, Z = Floor Z (down)
	wobj.uframe.trans := weld_start;
	wobj.uframe.rot.q1 := cos_half;
	wobj.uframe.rot.q2 := 0;
	wobj.uframe.rot.q3 := 0;
	wobj.uframe.rot.q4 := sin_half;

	! Object frame: identity (no additional offset)
	wobj.oframe.trans.x := 0;
	wobj.oframe.trans.y := 0;
	wobj.oframe.trans.z := 0;
	wobj.oframe.rot.q1 := 1;
	wobj.oframe.rot.q2 := 0;
	wobj.oframe.rot.q3 := 0;
	wobj.oframe.rot.q4 := 0;

	TPWrite "[WELD] Created WObj at [" + NumToStr(weld_start.x, 1) + ", "
	                                    + NumToStr(weld_start.y, 1) + ", "
	                                    + NumToStr(weld_start.z, 1) + "]";
	TPWrite "[WELD] WObj X+ direction: " + NumToStr(angle_deg, 2) + " deg from Floor X+";
ENDPROC

! ----------------------------------------
! Move Gantry to Weld Start Position
! ----------------------------------------
! Moves gantry to center line start with correct R-axis angle
! Robot joints are preserved (robots don't move)
PROC MoveGantryToWeldStart()
	VAR jointtarget current_jt;
	VAR jointtarget target_jt;
	VAR pos gantry_target;
	VAR iodev gantry_log;

	! v1.9.12: Detailed logging to diagnose linked motor error
	Open "HOME:/gantry_move_debug.txt", gantry_log \Write;
	Write gantry_log, "MoveGantryToWeldStart (" + TASK1_VERSION + ") " + CDate() + " " + CTime();

	TPWrite "[WELD] Moving gantry to weld start...";

	! Get current joint positions (preserve robot joints)
	current_jt := CJointT();
	Write gantry_log, "CJointT: X1=" + NumToStr(current_jt.extax.eax_a,1) + " X2=" + NumToStr(current_jt.extax.eax_f,1);

	! Calculate gantry target from center start (Floor -> Physical)
	gantry_target := CalcGantryFromFloor(weld_center_start);
	Write gantry_log, "Target: X=" + NumToStr(gantry_target.x,1) + " Y=" + NumToStr(gantry_target.y,1) + " Z=" + NumToStr(gantry_target.z,1);

	! Create target joint (keep robot joints, set gantry position)
	target_jt := current_jt;
	target_jt.extax.eax_a := gantry_target.x;  ! Gantry X1
	target_jt.extax.eax_b := gantry_target.y;  ! Gantry Y
	target_jt.extax.eax_c := gantry_target.z;  ! Gantry Z
	target_jt.extax.eax_d := weld_center_angle; ! Gantry R
	! v1.9.16: Set X2 to same value as X1 (linked motor requirement)
	target_jt.extax.eax_f := gantry_target.x;

	Write gantry_log, "Command: eax_a=" + NumToStr(target_jt.extax.eax_a,1) + " eax_f=" + NumToStr(target_jt.extax.eax_f,1);
	Write gantry_log, "Calling MoveAbsJ...";
	Close gantry_log;

	TPWrite "[WELD] Gantry target: [" + NumToStr(gantry_target.x, 1) + ", "
	                                   + NumToStr(gantry_target.y, 1) + ", "
	                                   + NumToStr(gantry_target.z, 1) + ", R="
	                                   + NumToStr(weld_center_angle, 2) + "]";

	! Move gantry (robot joints stay same)
	MoveAbsJ target_jt, v500, fine, tool0;

	! Update WobjGantry after gantry move
	UpdateGantryWobj;

	TPWrite "[WELD] Gantry at weld start position";
ENDPROC

! ----------------------------------------
! Move Robot1 to Weld Ready Position
! ----------------------------------------
! Moves Robot1 to weld position with 2-step approach
! v1.9.19: Step1 - MoveAbsJ to safe joint position
!          Step2 - MoveJ to wobj0 target position
PROC MoveRobot1ToWeldReady()
	VAR robtarget weld_target;
	VAR jointtarget safe_jt;
	VAR jointtarget current_jt;

	TPWrite "[WELD] Moving Robot1 to weld ready...";

	! Get current gantry position (Robot1 is gantry-configured)
	current_jt := CJointT();

	! Step 1: Move to safe JOINT position first
	! Robot joints: [0, -10, -50, 0, -30, 0]
	safe_jt := current_jt;  ! Keep gantry extax
	safe_jt.robax.rax_1 := 0;
	safe_jt.robax.rax_2 := -10;
	safe_jt.robax.rax_3 := -50;
	safe_jt.robax.rax_4 := 0;
	safe_jt.robax.rax_5 := -30;
	safe_jt.robax.rax_6 := 0;
	TPWrite "[WELD] R1 Step1: MoveAbsJ to safe joints";
	MoveAbsJ safe_jt, v100, fine, tool0;

	! Step 2: Move to WobjGantry target position
	! v1.9.22: Corrected WobjGantry coords from user jog data
	! User jog at X=-4500: wobj0 Y=110.59, Z=2026.89
	! WobjGantry = [0, 111, -73] (Z = 2026.89 - 2100)
	current_jt := CJointT();  ! Re-read after move
	UpdateGantryWobj;
	weld_target.trans.x := 0;
	weld_target.trans.y := 111;
	weld_target.trans.z := -73;
	weld_target.rot.q1 := WELD_R1_ORIENT_Q1;
	weld_target.rot.q2 := WELD_R1_ORIENT_Q2;
	weld_target.rot.q3 := WELD_R1_ORIENT_Q3;
	weld_target.rot.q4 := WELD_R1_ORIENT_Q4;
	weld_target.robconf.cf1 := 0;
	weld_target.robconf.cf4 := 0;
	weld_target.robconf.cf6 := 0;
	weld_target.robconf.cfx := 0;
	weld_target.extax := current_jt.extax;

	TPWrite "[WELD] R1 Step2: MoveJ to WobjGantry [0, 111, -73]";
	MoveJ weld_target, v100, fine, tWeld1\WObj:=WobjGantry;

	TPWrite "[WELD] Robot1 ready at weld position (tWeld1)";
ENDPROC

! ----------------------------------------
! Signal Robot2 to Move to Weld Ready
! ----------------------------------------
! Sets sync flag and waits for Robot2 to be ready
PROC WaitForRobot2WeldReady()
	TPWrite "[WELD] Waiting for Robot2 weld ready...";

	! Signal Robot2 to move to weld position
	t1_weld_start := TRUE;
	t2_weld_ready := FALSE;

	! Wait for Robot2 ready signal
	WHILE NOT t2_weld_ready DO
		WaitTime 0.1;
	ENDWHILE

	TPWrite "[WELD] Robot2 ready!";
ENDPROC

! ----------------------------------------
! Move Gantry Along Center Line (Welding)
! ----------------------------------------
! Moves gantry from start to end of center line
! Robots maintain position in their respective WObj (weld posture maintained)
PROC WeldAlongCenterLine()
	VAR jointtarget current_jt;
	VAR jointtarget end_jt;
	VAR pos gantry_end;

	TPWrite "[WELD] Starting weld along center line...";

	! Get current joint positions
	current_jt := CJointT();

	! Calculate gantry end position (Floor -> Physical)
	gantry_end := CalcGantryFromFloor(weld_center_end);

	! Create end joint target (keep robot joints, change gantry XY)
	end_jt := current_jt;
	end_jt.extax.eax_a := gantry_end.x;  ! Gantry X1
	end_jt.extax.eax_b := gantry_end.y;  ! Gantry Y
	! v1.9.16: Set X2 to same value as X1 (linked motor requirement)
	end_jt.extax.eax_f := gantry_end.x;
	! Z and R stay the same

	TPWrite "[WELD] Welding to [" + NumToStr(gantry_end.x, 1) + ", "
	                               + NumToStr(gantry_end.y, 1) + "]";
	TPWrite "[WELD] Speed: v100";

	! Move gantry along center line (robots stay in weld posture)
	! Speed: v100 (modify ConfigModule WELD_SPEED for future use)
	! v1.9.13: Use tool0 for testing
	MoveAbsJ end_jt, v100, fine, tool0;

	TPWrite "[WELD] Weld complete!";
ENDPROC

! ----------------------------------------
! Execute Complete Weld Sequence
! ----------------------------------------
! Main entry point for weld sequence
! Steps:
!   1. Calculate center line from weld lines
!   2. Move gantry to center start with R-axis aligned
!   3. Create weld WObjs for both robots
!   4. Move robots to weld ready positions
!   5. Execute weld (gantry moves, robots maintain posture)
PROC ExecuteWeldSequence()
	VAR pos r1_start;
	VAR pos r1_end;
	VAR pos r2_start;
	VAR pos r2_end;
	VAR iodev weld_logfile;
	VAR jointtarget current_jt;
	VAR num x1_val;
	VAR num x2_val;
	VAR num sync_distance;

	! v1.9.12: Added file logging for debugging
	Open "HOME:/weld_sequence.txt", weld_logfile \Write;
	Write weld_logfile, "Weld Sequence Log (" + TASK1_VERSION + ") Date=" + CDate() + " Time=" + CTime();

	TPWrite "========================================";
	TPWrite "[WELD] v1.9.12 Weld Sequence Start";
	TPWrite "========================================";

	! Log current gantry position
	current_jt := CJointT();
	x1_val := current_jt.extax.eax_a;
	x2_val := current_jt.extax.eax_f;
	sync_distance := x1_val - x2_val;
	Write weld_logfile, "Start extax: X1=" + NumToStr(x1_val,1) + " X2=" + NumToStr(x2_val,1) + " diff=" + NumToStr(sync_distance,1);

	! v1.9.12: X1/X2 are physically same axis (linked motors)
	! eax_f reported value may be stale software state - not physical difference
	! Solution: Just log the discrepancy, don't try to physically sync
	IF Abs(sync_distance) > 1 THEN
		Write weld_logfile, "NOTE: eax_f state mismatch (software state, not physical)";
		Write weld_logfile, "Physical axis position is eax_a=" + NumToStr(x1_val,1);
	ENDIF

	! Reset sync flags
	t1_weld_start := FALSE;
	t1_weld_done := FALSE;
	t2_weld_ready := FALSE;
	Write weld_logfile, "Step0: Sync flags reset";

	! Read weld line positions from ConfigModule
	r1_start.x := WELD_R1_START_X;
	r1_start.y := WELD_R1_START_Y;
	r1_start.z := WELD_R1_START_Z;
	r1_end.x := WELD_R1_END_X;
	r1_end.y := WELD_R1_END_Y;
	r1_end.z := WELD_R1_END_Z;
	r2_start.x := WELD_R2_START_X;
	r2_start.y := WELD_R2_START_Y;
	r2_start.z := WELD_R2_START_Z;
	r2_end.x := WELD_R2_END_X;
	r2_end.y := WELD_R2_END_Y;
	r2_end.z := WELD_R2_END_Z;

	Write weld_logfile, "R1 Line: [" + NumToStr(r1_start.x, 0) + "," + NumToStr(r1_start.y, 0) + "," + NumToStr(r1_start.z, 0) + "]";
	Write weld_logfile, "R2 Line: [" + NumToStr(r2_start.x, 0) + "," + NumToStr(r2_start.y, 0) + "," + NumToStr(r2_start.z, 0) + "]";
	TPWrite "[WELD] R1 Line: [" + NumToStr(r1_start.x, 0) + "," + NumToStr(r1_start.y, 0) + "," + NumToStr(r1_start.z, 0) + "] -> ["
	                             + NumToStr(r1_end.x, 0) + "," + NumToStr(r1_end.y, 0) + "," + NumToStr(r1_end.z, 0) + "]";
	TPWrite "[WELD] R2 Line: [" + NumToStr(r2_start.x, 0) + "," + NumToStr(r2_start.y, 0) + "," + NumToStr(r2_start.z, 0) + "] -> ["
	                             + NumToStr(r2_end.x, 0) + "," + NumToStr(r2_end.y, 0) + "," + NumToStr(r2_end.z, 0) + "]";

	! Step 1: Calculate center line
	Write weld_logfile, "Step1: CalcCenterLine START";
	CalcCenterLine;
	Write weld_logfile, "Step1: CalcCenterLine DONE";

	! Step 2: Move gantry to weld start position
	Write weld_logfile, "Step2: MoveGantryToWeldStart START";
	MoveGantryToWeldStart;
	current_jt := CJointT();
	Write weld_logfile, "Step2: MoveGantryToWeldStart DONE - X1=" + NumToStr(current_jt.extax.eax_a,1) + " X2=" + NumToStr(current_jt.extax.eax_f,1);

	! Step 3: Create weld WObjs
	Write weld_logfile, "Step3: CreateWeldWobj START";
	CreateWeldWobj r1_start, r1_end, WobjWeldR1;
	CreateWeldWobj r2_start, r2_end, WobjWeldR2;
	Write weld_logfile, "Step3: CreateWeldWobj DONE";

	! Step 4: Move robots to weld ready
	Write weld_logfile, "Step4a: MoveRobot1ToWeldReady START";
	MoveRobot1ToWeldReady;
	Write weld_logfile, "Step4a: MoveRobot1ToWeldReady DONE";

	Write weld_logfile, "Step4b: WaitForRobot2WeldReady START";
	WaitForRobot2WeldReady;
	Write weld_logfile, "Step4b: WaitForRobot2WeldReady DONE";

	! Step 5: Execute weld (gantry moves along center line)
	Write weld_logfile, "Step5: WeldAlongCenterLine START";
	WeldAlongCenterLine;
	Write weld_logfile, "Step5: WeldAlongCenterLine DONE";

	! Signal completion
	t1_weld_done := TRUE;

	! v1.9.20: Step 6 - Return robots to safe position
	Write weld_logfile, "Step6: ReturnToSafePosition START";
	ReturnRobot1ToSafe;
	Write weld_logfile, "Step6: ReturnToSafePosition DONE";

	! v1.9.20: Step 7 - Return gantry to HOME
	Write weld_logfile, "Step7: ReturnGantryToHome START";
	ReturnGantryToHome;
	Write weld_logfile, "Step7: ReturnGantryToHome DONE";

	Write weld_logfile, "Weld Sequence COMPLETE at " + CTime();
	Close weld_logfile;

	TPWrite "========================================";
	TPWrite "[WELD] Weld Sequence Complete!";
	TPWrite "========================================";
ENDPROC

! ----------------------------------------
! Return Robot1 to Safe Position
! ----------------------------------------
! v1.9.20: Move Robot1 to safe joint position after weld
PROC ReturnRobot1ToSafe()
	VAR jointtarget safe_jt;

	TPWrite "[WELD] Returning Robot1 to safe position...";

	! Get current position and move to safe joints
	safe_jt := CJointT();
	safe_jt.robax.rax_1 := 0;
	safe_jt.robax.rax_2 := -10;
	safe_jt.robax.rax_3 := -50;
	safe_jt.robax.rax_4 := 0;
	safe_jt.robax.rax_5 := -30;
	safe_jt.robax.rax_6 := 0;
	MoveAbsJ safe_jt, v100, fine, tool0;

	TPWrite "[WELD] Robot1 at safe position";
ENDPROC

! ----------------------------------------
! Return Gantry to HOME Position
! ----------------------------------------
! v1.9.20: Move gantry to HOME [0,0,0,0] after weld
PROC ReturnGantryToHome()
	VAR jointtarget home_jt;

	TPWrite "[WELD] Returning gantry to HOME...";

	! Get current position
	home_jt := CJointT();

	! Set gantry to HOME [0,0,0,0]
	home_jt.extax.eax_a := 0;  ! X1
	home_jt.extax.eax_b := 0;  ! Y
	home_jt.extax.eax_c := 0;  ! Z
	home_jt.extax.eax_d := 0;  ! R
	home_jt.extax.eax_f := 0;  ! X2 (linked motor)

	MoveAbsJ home_jt, v500, fine, tool0;

	TPWrite "[WELD] Gantry at HOME [0,0,0,0]";
ENDPROC

! ========================================
! Edge-based Weld Sequence Functions (v2.0.0)
! ========================================
! Ported from PlanA Head_MoveControl.mod
! Calculates center line from 4 edge points and determines R-axis angle

! ----------------------------------------
! Calculate Center Line from Edge Points
! ----------------------------------------
! Reads EDGE_START1/2, EDGE_END1/2 from ConfigModule
! Calculates calcPosStart, calcPosEnd as averages
PROC CalcCenterFromEdges()
	TPWrite "[EDGE] Calculating center line from edges...";

	! Calculate center line start (average of edgeStart{1} and edgeStart{2})
	calcPosStart.x := (EDGE_START1_X + EDGE_START2_X) / 2;
	calcPosStart.y := (EDGE_START1_Y + EDGE_START2_Y) / 2;
	calcPosStart.z := (EDGE_START1_Z + EDGE_START2_Z) / 2;

	! Calculate center line end (average of edgeEnd{1} and edgeEnd{2})
	calcPosEnd.x := (EDGE_END1_X + EDGE_END2_X) / 2;
	calcPosEnd.y := (EDGE_END1_Y + EDGE_END2_Y) / 2;
	calcPosEnd.z := (EDGE_END1_Z + EDGE_END2_Z) / 2;

	TPWrite "[EDGE] Edge Start 1: [" + NumToStr(EDGE_START1_X,0) + ","
	        + NumToStr(EDGE_START1_Y,0) + "," + NumToStr(EDGE_START1_Z,0) + "]";
	TPWrite "[EDGE] Edge Start 2: [" + NumToStr(EDGE_START2_X,0) + ","
	        + NumToStr(EDGE_START2_Y,0) + "," + NumToStr(EDGE_START2_Z,0) + "]";
	TPWrite "[EDGE] Edge End 1: [" + NumToStr(EDGE_END1_X,0) + ","
	        + NumToStr(EDGE_END1_Y,0) + "," + NumToStr(EDGE_END1_Z,0) + "]";
	TPWrite "[EDGE] Edge End 2: [" + NumToStr(EDGE_END2_X,0) + ","
	        + NumToStr(EDGE_END2_Y,0) + "," + NumToStr(EDGE_END2_Z,0) + "]";
	TPWrite "[EDGE] Center Start: [" + NumToStr(calcPosStart.x,1) + ","
	        + NumToStr(calcPosStart.y,1) + "," + NumToStr(calcPosStart.z,1) + "]";
	TPWrite "[EDGE] Center End: [" + NumToStr(calcPosEnd.x,1) + ","
	        + NumToStr(calcPosEnd.y,1) + "," + NumToStr(calcPosEnd.z,1) + "]";
ENDPROC

! ----------------------------------------
! Define Weld Line (R-axis Calculation)
! ----------------------------------------
! Ported from PlanA rDefineWobjWeldLine
! Calculates R-axis angle and determines bRobSwap
PROC DefineWeldLine()
	VAR num dx;
	VAR num dy;
	VAR num dz;
	VAR pos tempPos;

	TPWrite "[WELD] Defining weld line...";

	! Calculate direction vector
	dx := calcPosEnd.x - calcPosStart.x;
	dy := calcPosEnd.y - calcPosStart.y;
	dz := calcPosEnd.z - calcPosStart.z;

	! Calculate weld line length
	calcLengthWeldLine := Sqrt(dx*dx + dy*dy + dz*dz);

	! Calculate R-axis angle (ATan2 gives angle from X+ axis in degrees)
	! Floor coordinate: X+ = gantry forward, Y+ = left
	nAngleRzStore := ATan2(dy, dx);

	! Determine bRobSwap: TRUE when angle at or beyond +/-90deg (buffer/orient select)
	IF (nAngleRzStore <= -90 OR nAngleRzStore >= 90) THEN
		bRobSwap := TRUE;
		shared_bRobSwap := TRUE;
		TPWrite "[WELD] bRobSwap = TRUE (raw R=" + NumToStr(nAngleRzStore,1) + " deg)";

		! Swap start/end only when strictly outside +/-90deg (PlanC NormalizeAngle strict >)
		! At exactly +/-90deg: bRobSwap=TRUE for buffer, but no swap needed (within R limit)
		IF (nAngleRzStore < -90 OR nAngleRzStore > 90) THEN
			tempPos := calcPosStart;
			calcPosStart := calcPosEnd;
			calcPosEnd := tempPos;
			dx := calcPosEnd.x - calcPosStart.x;
			dy := calcPosEnd.y - calcPosStart.y;
			nAngleRzStore := ATan2(dy, dx);
			TPWrite "[WELD] Swapped start/end -> R=" + NumToStr(nAngleRzStore,1) + " deg";
		ENDIF
	ELSE
		bRobSwap := FALSE;
		shared_bRobSwap := FALSE;
		TPWrite "[WELD] bRobSwap = FALSE (R=" + NumToStr(nAngleRzStore,1) + " deg)";
	ENDIF

	! Calculate robot offset length
	IF calcLengthWeldLine < 20 THEN
		calcOffsetLengthBuffer := 10;
	ELSE
		calcOffsetLengthBuffer := 10;  ! Default offset for now
	ENDIF

	TPWrite "[WELD] R-axis angle: " + NumToStr(nAngleRzStore, 2) + " deg";
	TPWrite "[WELD] Weld length: " + NumToStr(calcLengthWeldLine, 1) + " mm";
ENDPROC

! ----------------------------------------
! Floor to Physical Coordinate Conversion
! ----------------------------------------
! Ported from PlanA fnCoordToJoint
! Converts Floor coordinates to Physical gantry coordinates
FUNC pos FloorToPhysical(pos floor_pos)
	VAR pos physical;

	! PlanA conversion formula:
	! Physical = HOME +/- (Floor - FloorHome)
	! FloorHome = [9500, 5300, 2100]
	physical.x := HOME_GANTRY_X + (floor_pos.x - 9500);   ! X: addition
	physical.y := HOME_GANTRY_Y - (floor_pos.y - 5300);   ! Y: subtraction (inverted)
	physical.z := HOME_GANTRY_Z - (floor_pos.z - 2100);   ! Z: subtraction (inverted)

	! Apply limits
	IF physical.x < nLimitX_Negative THEN
		physical.x := nLimitX_Negative;
	ENDIF
	IF physical.x > nLimitX_Positive THEN
		physical.x := nLimitX_Positive;
	ENDIF
	IF physical.y < nLimitY_Negative THEN
		physical.y := nLimitY_Negative;
	ENDIF
	IF physical.y > nLimitY_Positive THEN
		physical.y := nLimitY_Positive;
	ENDIF
	IF physical.z < nLimitZ_Negative THEN
		physical.z := nLimitZ_Negative;
	ENDIF
	IF physical.z > nLimitZ_Positive THEN
		physical.z := nLimitZ_Positive;
	ENDIF

	RETURN physical;
ENDFUNC

! ----------------------------------------
! Physical to Floor Coordinate Conversion
! ----------------------------------------
! Inverse of FloorToPhysical
! Converts Physical gantry coordinates to Floor coordinates
FUNC pos PhysicalToFloor(pos physical_pos)
	VAR pos floor;

	! Inverse of FloorToPhysical formula:
	! Floor = FloorHome +/- (Physical - HOME)
	! FloorHome = [9500, 5300, 2100]
	floor.x := 9500 + (physical_pos.x - HOME_GANTRY_X);   ! X: addition
	floor.y := 5300 - (physical_pos.y - HOME_GANTRY_Y);   ! Y: subtraction (inverted)
	floor.z := 2100 - (physical_pos.z - HOME_GANTRY_Z);   ! Z: subtraction (inverted)

	RETURN floor;
ENDFUNC

! ----------------------------------------
! Move Gantry to Weld Position
! ----------------------------------------
! Uses calculated calcPosStart and nAngleRzStore to position gantry
PROC MoveGantryToWeldPosition()
	VAR jointtarget current_jt;
	VAR jointtarget target_jt;
	VAR pos gantry_physical;
	VAR pos gantry_floor;
	VAR num target_r;
	VAR num offset_floor_x;
	VAR num offset_floor_y;

	TPWrite "[WELD] Moving gantry to weld position...";

	! Get current position
	current_jt := CJointT();
	target_jt := current_jt;

	! Debug: Show current X1/X2 position
	TPWrite "[DEBUG] Current X1=" + NumToStr(current_jt.extax.eax_a,1)
	       + " X2=" + NumToStr(current_jt.extax.eax_f,1)
	       + " diff=" + NumToStr(current_jt.extax.eax_a - current_jt.extax.eax_f,1);

	! Check linked motor sync (max_offset = 2mm in MOC.cfg)
	! X1 and X2 MUST move together - cannot sync independently
	IF Abs(current_jt.extax.eax_a - current_jt.extax.eax_f) > 2 THEN
		TPWrite "[ERROR] X1/X2 not synced (diff > 2mm)!";
		TPWrite "[ERROR] Linked motor requires X1=X2 (max offset: 2mm)";
		TPWrite "[ERROR] Please restart controller or manually jog to sync";
		TPWrite "[ERROR] Current diff: " + NumToStr(Abs(current_jt.extax.eax_a - current_jt.extax.eax_f),1) + "mm";
		Stop;
	ENDIF

	! Calculate R-axis (nAngleRzStore already +/-90deg after DefineWeldLine swap)
	target_r := HOME_GANTRY_R - nAngleRzStore;

	! v1.9.63c: Safety clamp only (swap in DefineWeldLine guarantees +/-90deg)
	IF target_r > nLimitR_Positive THEN
		target_r := nLimitR_Positive;
	ELSEIF target_r < nLimitR_Negative THEN
		target_r := nLimitR_Negative;
	ENDIF
	TPWrite "[WELD] R-axis: " + NumToStr(target_r,1) + " deg";

	! v1.9.64: Fixed TCP offset Floor calculation
	! WobjGantry = Physical coords with identity rotation (UpdateGantryWobj L1460-1466)
	! R-axis rotates robot base, NOT WobjGantry frame
	! Robot TCP in WobjGantry [X_wg, Y_wg] maps to Physical as [X_wg, Y_wg] (identity)
	! Physical-to-Floor: X same direction, Y INVERTED (FloorToPhysical L3720)
	! Therefore: offset_floor = [X_wg, -Y_wg] (no R rotation, Y negated)
	offset_floor_x := MODE2_TCP_OFFSET_R1_X;
	offset_floor_y := -MODE2_TCP_OFFSET_R1_Y;

	! Calculate gantry Floor position (gantry = weld_center - tcp_offset)
	! Gantry must be offset so that TCP reaches the weld center
	gantry_floor := calcPosStart;
	gantry_floor.x := gantry_floor.x - offset_floor_x;
	gantry_floor.y := gantry_floor.y - offset_floor_y;
	! Z offset: Gantry must be ABOVE weld so TCP can reach down
	! Apply in Floor coordinates BEFORE FloorToPhysical to avoid premature limit clamping
	! (v1.9.33 fix: was applied after FloorToPhysical causing 300mm error at low Z)
	gantry_floor.z := gantry_floor.z + WELD_R1_TCP_Z_OFFSET;

	TPWrite "[WELD] TCP offset (Floor): X=" + NumToStr(offset_floor_x,1) + " Y=" + NumToStr(offset_floor_y,1) + " Z=" + NumToStr(WELD_R1_TCP_Z_OFFSET,0);

	! Convert gantry Floor position to Physical coordinates
	! FloorToPhysical applies limits internally
	gantry_physical := FloorToPhysical(gantry_floor);

	! Set gantry target
	target_jt.extax.eax_a := gantry_physical.x;  ! X1
	target_jt.extax.eax_b := gantry_physical.y;  ! Y
	target_jt.extax.eax_c := gantry_physical.z;  ! Z
	target_jt.extax.eax_d := target_r;            ! R
	target_jt.extax.eax_f := gantry_physical.x;  ! X2 = X1 (linked motor)

	TPWrite "[WELD] Gantry target (Physical):";
	TPWrite "  X1=" + NumToStr(gantry_physical.x,1) + " mm";
	TPWrite "  Y=" + NumToStr(gantry_physical.y,1) + " mm";
	TPWrite "  Z=" + NumToStr(gantry_physical.z,1) + " mm";
	TPWrite "  R=" + NumToStr(target_r,1) + " deg";

	! Debug: Show target extax values
	TPWrite "[DEBUG] Target eax_a=" + NumToStr(target_jt.extax.eax_a,1)
	       + " eax_f=" + NumToStr(target_jt.extax.eax_f,1);

	! Move gantry
	TPWrite "[DEBUG] Calling MoveAbsJ...";
	MoveAbsJ target_jt, v500, fine, tool0;

	! Update WobjGantry after movement
	UpdateGantryWobj;

	TPWrite "[WELD] Gantry at weld position";
ENDPROC

! ----------------------------------------
! CheckLinkedMotorSync: Verify X1/X2 are synchronized
! ----------------------------------------
! Linked motor configuration (MOC.cfg):
!   - ELM_X is follower to M1DM3 (max_offset = 2mm)
!   - X1 (eax_a) and X2 (eax_f) must move together
!   - Cannot be synced from RAPID - must restart controller
PROC CheckLinkedMotorSync()
	VAR jointtarget jt;
	VAR num diff;

	jt := CJointT();
	diff := Abs(jt.extax.eax_a - jt.extax.eax_f);

	TPWrite "----------------------------------------";
	TPWrite "[LINKED MOTOR] Status Check";
	TPWrite "  X1 (Master): " + NumToStr(jt.extax.eax_a,1) + " mm";
	TPWrite "  X2 (Follower): " + NumToStr(jt.extax.eax_f,1) + " mm";
	TPWrite "  Difference: " + NumToStr(diff,1) + " mm";
	TPWrite "  Max Allowed: 2 mm (MOC.cfg LINKED_M_PROCESS)";

	IF diff > 2 THEN
		TPWrite "[LINKED MOTOR] ERROR: Out of sync!";
		TPWrite "[LINKED MOTOR] Attempting auto-fix...";
		ForceLinkedMotorSync;
	ELSE
		TPWrite "[LINKED MOTOR] OK - In sync";
		TPWrite "----------------------------------------";
	ENDIF
ENDPROC

! ----------------------------------------
! Force Linked Motor Sync (v1.9.25)
! ----------------------------------------
! Attempts to fix X1/X2 software state mismatch
! by forcing eax_f := eax_a and performing MoveAbsJ
PROC ForceLinkedMotorSync()
	VAR jointtarget current_jt;
	VAR jointtarget sync_jt;
	VAR num x1_val;

	current_jt := CJointT();
	x1_val := current_jt.extax.eax_a;

	TPWrite "[SYNC] Forcing X2 := X1 (" + NumToStr(x1_val,1) + " mm)";

	! Create sync target: keep all values, but force eax_f = eax_a
	sync_jt := current_jt;
	sync_jt.extax.eax_f := x1_val;

	! Try MoveAbsJ with synced values
	TPWrite "[SYNC] Executing MoveAbsJ to sync software state...";

	MoveAbsJ sync_jt, v100, fine, tool0;

	! Verify sync
	current_jt := CJointT();
	IF Abs(current_jt.extax.eax_a - current_jt.extax.eax_f) <= 2 THEN
		TPWrite "[SYNC] SUCCESS - X1/X2 now synced!";
		TPWrite "  X1=" + NumToStr(current_jt.extax.eax_a,1);
		TPWrite "  X2=" + NumToStr(current_jt.extax.eax_f,1);
		TPWrite "----------------------------------------";
	ELSE
		TPWrite "[SYNC] FAILED - Still out of sync";
		TPWrite "[SYNC] Manual restart required";
		TPWrite "----------------------------------------";
		Stop;
	ENDIF
ERROR
	TPWrite "[SYNC] ERROR during MoveAbsJ: " + NumToStr(ERRNO,0);
	TPWrite "[SYNC] Manual restart required";
	TPWrite "----------------------------------------";
	Stop;
ENDPROC

! ----------------------------------------
! Test: Weld Sequence (stub)
! ----------------------------------------
! Placeholder for weld sequence testing
! TODO: Implement actual weld sequence with arc control
PROC TestWeldSequence()
	! PlanC Phase 1: Route "Weld" command to full edge-based weld sequence
	! Same flow as "EdgeWeld" command (Gantry + Robot1 + Robot2 sync + TraceWeldLine)
	TestFullWeldSequence;
ENDPROC

! ----------------------------------------
! Test: Edge to Weld Calculation Only (No Movement)
! ----------------------------------------
! Verifies calculation logic without MoveAbsJ
! Output: HOME:/edge_to_weld_calc.txt
PROC TestEdgeToWeldCalcOnly()
	VAR pos gantry_physical;
	VAR pos gantry_physical_raw;
	VAR pos gantry_floor;
	VAR num target_r;
	VAR iodev logfile;
	VAR num offset_floor_x;
	VAR num offset_floor_y;

	TPWrite "========================================";
	TPWrite "[TEST] Edge to Weld CALC ONLY v1.2";
	TPWrite "[TEST] + X/Y TCP Offset Support";
	TPWrite "[TEST] Log: HOME:/edge_to_weld_calc.txt";
	TPWrite "========================================";

	! Open log file
	Open "HOME:/edge_to_weld_calc.txt", logfile \Write;
	Write logfile, "========================================";
	Write logfile, "Edge to Weld Calculation Log";
	Write logfile, "Date: " + CDate() + " Time: " + CTime();
	Write logfile, "========================================";
	Write logfile, "";

	! Step 1: Calculate center from edges
	TPWrite "[CALC] Step 1: Calculate center line...";
	Write logfile, "[STEP 1] Calculate center from edges";
	CalcCenterFromEdges;

	! Step 2: Define weld line (R-axis calculation)
	TPWrite "[CALC] Step 2: Define weld line (R-axis)...";
	Write logfile, "[STEP 2] Define weld line (R-axis)";
	DefineWeldLine;

	! Step 3: Calculate gantry target (no movement)
	Write logfile, "[STEP 3] Calculate gantry physical target";
	Write logfile, "";

	! Log input parameters
	Write logfile, "--- INPUT: Edge Points (Floor) ---";
	Write logfile, "EDGE_START1: [" + NumToStr(EDGE_START1_X,1) + ", " + NumToStr(EDGE_START1_Y,1) + ", " + NumToStr(EDGE_START1_Z,1) + "]";
	Write logfile, "EDGE_START2: [" + NumToStr(EDGE_START2_X,1) + ", " + NumToStr(EDGE_START2_Y,1) + ", " + NumToStr(EDGE_START2_Z,1) + "]";
	Write logfile, "EDGE_END1:   [" + NumToStr(EDGE_END1_X,1) + ", " + NumToStr(EDGE_END1_Y,1) + ", " + NumToStr(EDGE_END1_Z,1) + "]";
	Write logfile, "EDGE_END2:   [" + NumToStr(EDGE_END2_X,1) + ", " + NumToStr(EDGE_END2_Y,1) + ", " + NumToStr(EDGE_END2_Z,1) + "]";
	Write logfile, "";

	! Log calculation results
	Write logfile, "--- RESULT: Center Line (Floor) ---";
	Write logfile, "calcPosStart: [" + NumToStr(calcPosStart.x,1) + ", " + NumToStr(calcPosStart.y,1) + ", " + NumToStr(calcPosStart.z,1) + "]";
	Write logfile, "calcPosEnd:   [" + NumToStr(calcPosEnd.x,1) + ", " + NumToStr(calcPosEnd.y,1) + ", " + NumToStr(calcPosEnd.z,1) + "]";
	Write logfile, "nAngleRzStore: " + NumToStr(nAngleRzStore,2) + " deg";
	Write logfile, "bRobSwap: " + ValToStr(bRobSwap);
	Write logfile, "calcLengthWeldLine: " + NumToStr(calcLengthWeldLine,1) + " mm";
	Write logfile, "";

	! Calculate R-axis (nAngleRzStore already +/-90deg after DefineWeldLine swap)
	target_r := HOME_GANTRY_R - nAngleRzStore;
	! v1.9.63c: Safety clamp only
	IF target_r > nLimitR_Positive THEN target_r := nLimitR_Positive; ENDIF
	IF target_r < nLimitR_Negative THEN target_r := nLimitR_Negative; ENDIF

	! Calculate X/Y TCP offsets rotated by gantry R-axis angle
	Write logfile, "--- X/Y TCP Offset Calculation ---";
	Write logfile, "MODE2_TCP_OFFSET_R1_X: " + NumToStr(MODE2_TCP_OFFSET_R1_X,1) + " mm";
	Write logfile, "MODE2_TCP_OFFSET_R1_Y: " + NumToStr(MODE2_TCP_OFFSET_R1_Y,1) + " mm";
	Write logfile, "nAngleRzStore (weld line): " + NumToStr(nAngleRzStore,2) + " deg";
	Write logfile, "target_r (gantry R): " + NumToStr(target_r,1) + " deg";
	Write logfile, "NOTE: Use target_r for rotation (actual gantry angle)";
	Write logfile, "NOTE: RAPID Cos/Sin use DEGREES directly!";
	offset_floor_x := MODE2_TCP_OFFSET_R1_X * Cos(target_r) - MODE2_TCP_OFFSET_R1_Y * Sin(target_r);
	offset_floor_y := MODE2_TCP_OFFSET_R1_X * Sin(target_r) + MODE2_TCP_OFFSET_R1_Y * Cos(target_r);
	Write logfile, "Rotated TCP offset (Floor):";
	Write logfile, "  offset_floor_x: " + NumToStr(offset_floor_x,1) + " mm";
	Write logfile, "  offset_floor_y: " + NumToStr(offset_floor_y,1) + " mm";
	Write logfile, "";

	! Calculate gantry Floor position (gantry = weld_center - tcp_offset)
	Write logfile, "--- Gantry Floor Position (with X/Y offset) ---";
	Write logfile, "calcPosStart (weld center): [" + NumToStr(calcPosStart.x,1) + ", " + NumToStr(calcPosStart.y,1) + ", " + NumToStr(calcPosStart.z,1) + "]";
	gantry_floor := calcPosStart;
	gantry_floor.x := gantry_floor.x - offset_floor_x;
	gantry_floor.y := gantry_floor.y - offset_floor_y;
	Write logfile, "gantry_floor (after X/Y offset): [" + NumToStr(gantry_floor.x,1) + ", " + NumToStr(gantry_floor.y,1) + ", " + NumToStr(gantry_floor.z,1) + "]";
	Write logfile, "";

	! Calculate FloorToPhysical (raw, before Z offset)
	gantry_physical_raw := FloorToPhysical(gantry_floor);
	Write logfile, "--- FloorToPhysical Conversion ---";
	Write logfile, "Formula: Physical = HOME + (Floor - FloorHome)";
	Write logfile, "  FloorHome = [9500, 5300, 2100]";
	Write logfile, "  HOME_GANTRY = [" + NumToStr(HOME_GANTRY_X,1) + ", " + NumToStr(HOME_GANTRY_Y,1) + ", " + NumToStr(HOME_GANTRY_Z,1) + "]";
	Write logfile, "";
	Write logfile, "gantry_floor: [" + NumToStr(gantry_floor.x,1) + ", " + NumToStr(gantry_floor.y,1) + ", " + NumToStr(gantry_floor.z,1) + "]";
	Write logfile, "gantry_physical_raw: [" + NumToStr(gantry_physical_raw.x,1) + ", " + NumToStr(gantry_physical_raw.y,1) + ", " + NumToStr(gantry_physical_raw.z,1) + "]";
	Write logfile, "";

	! Apply Z offset (SUBTRACT because Physical Z is inverse of Floor Z)
	! Gantry must be ABOVE weld so TCP can reach down
	gantry_physical := gantry_physical_raw;
	Write logfile, "--- Z Offset Calculation (CORRECTED) ---";
	Write logfile, "WELD_R1_TCP_Z_OFFSET: " + NumToStr(WELD_R1_TCP_Z_OFFSET,1) + " mm";
	Write logfile, "gantry_physical.z (before): " + NumToStr(gantry_physical.z,1) + " mm";
	Write logfile, "Formula: Gantry_Z = Raw_Z - TCP_OFFSET (subtract!)";
	gantry_physical.z := gantry_physical.z - WELD_R1_TCP_Z_OFFSET;
	Write logfile, "gantry_physical.z (after offset): " + NumToStr(gantry_physical.z,1) + " mm";
	Write logfile, "LIMIT_Z: [" + NumToStr(nLimitZ_Negative,1) + ", " + NumToStr(nLimitZ_Positive,1) + "] mm";
	IF gantry_physical.z < nLimitZ_Negative THEN
		gantry_physical.z := nLimitZ_Negative;
		Write logfile, "gantry_physical.z (limited to min): " + NumToStr(gantry_physical.z,1) + " mm";
	ENDIF
	IF gantry_physical.z > nLimitZ_Positive THEN
		gantry_physical.z := nLimitZ_Positive;
		Write logfile, "gantry_physical.z (limited to max): " + NumToStr(gantry_physical.z,1) + " mm";
	ENDIF
	Write logfile, "";

	! Log R-axis (already calculated above for X/Y offset rotation)
	Write logfile, "--- R-axis Summary ---";
	Write logfile, "HOME_GANTRY_R: " + NumToStr(HOME_GANTRY_R,1) + " deg";
	Write logfile, "nAngleRzStore: " + NumToStr(nAngleRzStore,2) + " deg";
	Write logfile, "target_r (final, with limits): " + NumToStr(target_r,1) + " deg";
	Write logfile, "LIMIT_R: [" + NumToStr(nLimitR_Negative,1) + ", " + NumToStr(nLimitR_Positive,1) + "] deg";
	Write logfile, "";

	! Final target summary
	Write logfile, "========================================";
	Write logfile, "FINAL GANTRY TARGET (Physical)";
	Write logfile, "========================================";
	Write logfile, "X1 (eax_a): " + NumToStr(gantry_physical.x,1) + " mm";
	Write logfile, "Y  (eax_b): " + NumToStr(gantry_physical.y,1) + " mm";
	Write logfile, "Z  (eax_c): " + NumToStr(gantry_physical.z,1) + " mm";
	Write logfile, "R  (eax_d): " + NumToStr(target_r,1) + " deg";
	Write logfile, "X2 (eax_f): " + NumToStr(gantry_physical.x,1) + " mm (=X1, linked)";
	Write logfile, "========================================";
	Write logfile, "";

	! Close log file
	Close logfile;

	! Display results on TP
	TPWrite "----------------------------------------";
	TPWrite "[INPUT] Edge Points (Floor):";
	TPWrite "  Start1: [" + NumToStr(EDGE_START1_X,0) + "," + NumToStr(EDGE_START1_Y,0) + "," + NumToStr(EDGE_START1_Z,0) + "]";
	TPWrite "  Start2: [" + NumToStr(EDGE_START2_X,0) + "," + NumToStr(EDGE_START2_Y,0) + "," + NumToStr(EDGE_START2_Z,0) + "]";
	TPWrite "  End1: [" + NumToStr(EDGE_END1_X,0) + "," + NumToStr(EDGE_END1_Y,0) + "," + NumToStr(EDGE_END1_Z,0) + "]";
	TPWrite "  End2: [" + NumToStr(EDGE_END2_X,0) + "," + NumToStr(EDGE_END2_Y,0) + "," + NumToStr(EDGE_END2_Z,0) + "]";
	TPWrite "----------------------------------------";
	TPWrite "[RESULT] Center (Floor):";
	TPWrite "  Start: [" + NumToStr(calcPosStart.x,1) + "," + NumToStr(calcPosStart.y,1) + "," + NumToStr(calcPosStart.z,1) + "]";
	TPWrite "  End: [" + NumToStr(calcPosEnd.x,1) + "," + NumToStr(calcPosEnd.y,1) + "," + NumToStr(calcPosEnd.z,1) + "]";
	TPWrite "[RESULT] R-axis: " + NumToStr(nAngleRzStore,2) + " deg";
	TPWrite "[RESULT] bRobSwap: " + ValToStr(bRobSwap);
	TPWrite "[RESULT] Weld Length: " + NumToStr(calcLengthWeldLine,1) + " mm";
	TPWrite "----------------------------------------";
	TPWrite "[OFFSET] TCP X/Y (rotated to Floor):";
	TPWrite "  X: " + NumToStr(offset_floor_x,1) + " mm, Y: " + NumToStr(offset_floor_y,1) + " mm";
	TPWrite "[TARGET] Gantry Physical (with offsets):";
	TPWrite "  X: " + NumToStr(gantry_physical.x,1) + " mm";
	TPWrite "  Y: " + NumToStr(gantry_physical.y,1) + " mm";
	TPWrite "  Z: " + NumToStr(gantry_physical.z,1) + " mm (limit:" + NumToStr(nLimitZ_Positive,0) + ")";
	TPWrite "  R: " + NumToStr(target_r,1) + " deg";
	TPWrite "========================================";
	TPWrite "[TEST] Log saved: HOME:/edge_to_weld_calc.txt";
	TPWrite "========================================";
ENDPROC

! ----------------------------------------
! Test: Edge to Weld Position
! ----------------------------------------
! Complete test of edge input to gantry positioning
PROC TestEdgeToWeld()
	VAR jointtarget actual_jt;
	VAR robtarget actual_tcp_wobj;
	VAR robtarget actual_tcp_gantry;
	VAR pos target_floor;
	VAR pos gantry_physical;
	VAR pos gantry_floor;
	VAR pos calc_tcp_floor;
	VAR num target_r;
	VAR num offset_floor_x;
	VAR num offset_floor_y;
	VAR num err_x;
	VAR num err_y;
	VAR num err_z;
	VAR num err_total;
	VAR iodev logfile;

	TPWrite "========================================";
	TPWrite "[TEST] Edge to Weld Position Test v2.3.0";
	TPWrite "[TEST] + TCP Tracking (Gantry-based)";
	TPWrite "========================================";

	! Step 0: Check linked motor sync (X1/X2)
	TPWrite "[TEST] Step 0: Check linked motor sync...";
	CheckLinkedMotorSync;

	! Step 1: Calculate center from edges
	TPWrite "[TEST] Step 1: Calculate center line...";
	CalcCenterFromEdges;

	! Step 2: Define weld line (R-axis calculation)
	TPWrite "[TEST] Step 2: Define weld line (R-axis)...";
	DefineWeldLine;

	! Step 3: Display calculated results
	TPWrite "----------------------------------------";
	TPWrite "[RESULT] Center Start: [" + NumToStr(calcPosStart.x,1) + ","
	        + NumToStr(calcPosStart.y,1) + "," + NumToStr(calcPosStart.z,1) + "]";
	TPWrite "[RESULT] Center End: [" + NumToStr(calcPosEnd.x,1) + ","
	        + NumToStr(calcPosEnd.y,1) + "," + NumToStr(calcPosEnd.z,1) + "]";
	TPWrite "[RESULT] R-axis: " + NumToStr(nAngleRzStore,2) + " deg";
	TPWrite "[RESULT] bRobSwap: " + ValToStr(bRobSwap);
	TPWrite "[RESULT] Weld Length: " + NumToStr(calcLengthWeldLine,1) + " mm";
	TPWrite "----------------------------------------";

	! Step 4: Move gantry to weld position
	TPWrite "[TEST] Step 4: Move gantry to weld position...";
	MoveGantryToWeldPosition;

	! Step 5: Verify gantry position
	actual_jt := CJointT();
	TPWrite "----------------------------------------";
	TPWrite "[VERIFY] Actual Gantry Position:";
	TPWrite "  X1=" + NumToStr(actual_jt.extax.eax_a,1) + " mm";
	TPWrite "  Y=" + NumToStr(actual_jt.extax.eax_b,1) + " mm";
	TPWrite "  Z=" + NumToStr(actual_jt.extax.eax_c,1) + " mm";
	TPWrite "  R=" + NumToStr(actual_jt.extax.eax_d,1) + " deg";
	TPWrite "  X2=" + NumToStr(actual_jt.extax.eax_f,1) + " mm";

	! Step 6: TCP Tracking Verification (Gantry-based calculation)
	TPWrite "----------------------------------------";
	TPWrite "[TCP] Step 6: TCP Tracking Verification";

	! Target: calcPosStart (weld start position in Floor coordinates)
	target_floor := calcPosStart;
	TPWrite "[TCP] Target Weld (Floor): [" + NumToStr(target_floor.x,1) + ", "
	        + NumToStr(target_floor.y,1) + ", " + NumToStr(target_floor.z,1) + "]";

	! Get actual gantry position and convert to Floor
	gantry_physical.x := actual_jt.extax.eax_a;
	gantry_physical.y := actual_jt.extax.eax_b;
	gantry_physical.z := actual_jt.extax.eax_c;
	target_r := actual_jt.extax.eax_d;
	gantry_floor := PhysicalToFloor(gantry_physical);
	TPWrite "[TCP] Gantry (Floor): [" + NumToStr(gantry_floor.x,1) + ", "
	        + NumToStr(gantry_floor.y,1) + ", " + NumToStr(gantry_floor.z,1) + "]";
	TPWrite "[TCP] Gantry R: " + NumToStr(target_r,1) + " deg";

	! Calculate TCP offset rotated by R-axis angle
	! TCP offset in Floor coords = Rot(R) * [TCP_X, TCP_Y]
	offset_floor_x := MODE2_TCP_OFFSET_R1_X * Cos(target_r) - MODE2_TCP_OFFSET_R1_Y * Sin(target_r);
	offset_floor_y := MODE2_TCP_OFFSET_R1_X * Sin(target_r) + MODE2_TCP_OFFSET_R1_Y * Cos(target_r);
	TPWrite "[TCP] Rotated Offset: [" + NumToStr(offset_floor_x,1) + ", " + NumToStr(offset_floor_y,1) + "]";

	! Calculate expected TCP position in Floor coordinates
	! TCP_floor = Gantry_floor + Rotated_TCP_Offset
	calc_tcp_floor.x := gantry_floor.x + offset_floor_x;
	calc_tcp_floor.y := gantry_floor.y + offset_floor_y;
	calc_tcp_floor.z := gantry_floor.z - WELD_R1_TCP_Z_OFFSET;  ! Z: gantry above, TCP below
	TPWrite "[TCP] Calculated TCP (Floor): [" + NumToStr(calc_tcp_floor.x,1) + ", "
	        + NumToStr(calc_tcp_floor.y,1) + ", " + NumToStr(calc_tcp_floor.z,1) + "]";

	! Calculate tracking error (Target vs Calculated)
	err_x := calc_tcp_floor.x - target_floor.x;
	err_y := calc_tcp_floor.y - target_floor.y;
	err_z := calc_tcp_floor.z - target_floor.z;
	err_total := Sqrt(err_x*err_x + err_y*err_y + err_z*err_z);

	TPWrite "[TCP] Tracking Error (Calc vs Target):";
	TPWrite "  dX=" + NumToStr(err_x,2) + " mm";
	TPWrite "  dY=" + NumToStr(err_y,2) + " mm";
	TPWrite "  dZ=" + NumToStr(err_z,2) + " mm";
	TPWrite "  Total=" + NumToStr(err_total,2) + " mm";

	! Also read actual TCP in WobjGantry for reference
	UpdateGantryWobj;
	actual_tcp_gantry := CRobT(\Tool:=tWeld1\WObj:=WobjGantry);
	TPWrite "[TCP] Actual TCP (WobjGantry): [" + NumToStr(actual_tcp_gantry.trans.x,1) + ", "
	        + NumToStr(actual_tcp_gantry.trans.y,1) + ", " + NumToStr(actual_tcp_gantry.trans.z,1) + "]";

	! Log to file
	Open "HOME:/tcp_tracking.txt", logfile \Write;
	Write logfile, "TCP Tracking Log (v2.3) - " + CDate() + " " + CTime();
	Write logfile, "";
	Write logfile, "--- Target ---";
	Write logfile, "Weld Start (Floor): [" + NumToStr(target_floor.x,1) + ", " + NumToStr(target_floor.y,1) + ", " + NumToStr(target_floor.z,1) + "]";
	Write logfile, "";
	Write logfile, "--- Gantry Position ---";
	Write logfile, "Physical: X=" + NumToStr(gantry_physical.x,1) + " Y=" + NumToStr(gantry_physical.y,1) + " Z=" + NumToStr(gantry_physical.z,1) + " R=" + NumToStr(target_r,1);
	Write logfile, "Floor: [" + NumToStr(gantry_floor.x,1) + ", " + NumToStr(gantry_floor.y,1) + ", " + NumToStr(gantry_floor.z,1) + "]";
	Write logfile, "";
	Write logfile, "--- TCP Offset Calculation ---";
	Write logfile, "TCP Offset (raw): X=" + NumToStr(MODE2_TCP_OFFSET_R1_X,1) + " Y=" + NumToStr(MODE2_TCP_OFFSET_R1_Y,1);
	Write logfile, "TCP Offset (rotated by R=" + NumToStr(target_r,1) + "): [" + NumToStr(offset_floor_x,1) + ", " + NumToStr(offset_floor_y,1) + "]";
	Write logfile, "";
	Write logfile, "--- Calculated TCP Position ---";
	Write logfile, "TCP Floor (calc): [" + NumToStr(calc_tcp_floor.x,1) + ", " + NumToStr(calc_tcp_floor.y,1) + ", " + NumToStr(calc_tcp_floor.z,1) + "]";
	Write logfile, "";
	Write logfile, "--- Tracking Error ---";
	Write logfile, "dX=" + NumToStr(err_x,2) + " dY=" + NumToStr(err_y,2) + " dZ=" + NumToStr(err_z,2) + " Total=" + NumToStr(err_total,2) + " mm";
	Write logfile, "";
	Write logfile, "--- Robot TCP (reference) ---";
	Write logfile, "TCP in WobjGantry: [" + NumToStr(actual_tcp_gantry.trans.x,1) + ", " + NumToStr(actual_tcp_gantry.trans.y,1) + ", " + NumToStr(actual_tcp_gantry.trans.z,1) + "]";
	Close logfile;
	TPWrite "[TCP] Log saved: HOME:/tcp_tracking.txt";

	TPWrite "========================================";
	TPWrite "[TEST] Edge to Weld Position Test Complete";
	TPWrite "========================================";

	! Step 7: Return gantry to HOME
	TPWrite "";
	TPWrite "[TEST] Step 7: Returning to HOME...";
	ReturnGantryToHome;
	TPWrite "[TEST] Gantry returned to HOME [0,0,0,0]";
	TPWrite "========================================";
ENDPROC

! ----------------------------------------
! Test Multi-Angle: Test 0deg, 45deg, 90deg, -45deg (v2.4.0)
! ----------------------------------------
! Tests 4 different weld line angles to verify calculation accuracy
! Temporarily changes EDGE points, runs test, and logs results
PROC TestMultiAngle()
	VAR num orig_end1_x;
	VAR num orig_end1_y;
	VAR num orig_end2_x;
	VAR num orig_end2_y;
	VAR num test_angles{4};
	VAR num test_dx{4};
	VAR num test_dy{4};
	VAR num i;
	VAR iodev logfile;
	VAR jointtarget actual_jt;
	VAR pos gantry_physical;
	VAR pos gantry_floor;
	VAR pos target_floor;
	VAR pos calc_tcp_floor;
	VAR num target_r;
	VAR num offset_floor_x;
	VAR num offset_floor_y;
	VAR num err_x;
	VAR num err_y;
	VAR num err_z;
	VAR num err_total;
	VAR robtarget actual_tcp_gantry;

	TPWrite "========================================";
	TPWrite "[MULTI] Multi-Angle Test v2.4.0";
	TPWrite "========================================";

	! Save original edge points
	orig_end1_x := EDGE_END1_X;
	orig_end1_y := EDGE_END1_Y;
	orig_end2_x := EDGE_END2_X;
	orig_end2_y := EDGE_END2_Y;

	! Define test angles (degrees) and corresponding dx, dy for 500mm weld line
	! 0deg:   dx=500, dy=0    (horizontal X+)
	! 45deg:  dx=354, dy=354  (diagonal)
	! 90deg:  dx=0,   dy=500  (vertical Y+)
	! -45deg: dx=354, dy=-354 (diagonal X+, Y-)
	test_angles{1} := 0;
	test_dx{1} := 500;
	test_dy{1} := 0;
	test_angles{2} := 45;
	test_dx{2} := 354;
	test_dy{2} := 354;
	test_angles{3} := 90;
	test_dx{3} := 0;
	test_dy{3} := 500;
	test_angles{4} := -45;
	test_dx{4} := 354;
	test_dy{4} := -354;

	! Open log file
	Open "HOME:/multi_angle_test.txt", logfile \Write;
	Write logfile, "Multi-Angle Test Log (v2.4.0) - " + CDate() + " " + CTime();
	Write logfile, "";
	Write logfile, "Start Point (Floor): [" + NumToStr(EDGE_START1_X,0) + ", " + NumToStr(EDGE_START1_Y,0) + ", " + NumToStr(EDGE_START1_Z,0) + "]";
	Write logfile, "";
	Write logfile, "Angle | Expected R | Actual R | Error X | Error Y | Total (mm)";
	Write logfile, "------+-----------+----------+---------+---------+-----------";

	! Run tests for each angle
	FOR i FROM 1 TO 4 DO
		TPWrite "";
		TPWrite "----------------------------------------";
		TPWrite "[MULTI] Test " + NumToStr(i,0) + "/4: Angle = " + NumToStr(test_angles{i},0) + " deg";
		TPWrite "----------------------------------------";

		! Set edge end points for this angle
		! Robot1 side: center + dy/2
		! Robot2 side: center - dy/2
		EDGE_END1_X := EDGE_START1_X + test_dx{i};
		EDGE_END1_Y := EDGE_START1_Y + test_dy{i};
		EDGE_END2_X := EDGE_START2_X + test_dx{i};
		EDGE_END2_Y := EDGE_START2_Y + test_dy{i};

		TPWrite "[MULTI] Edge End: [" + NumToStr(EDGE_END1_X,0) + ", " + NumToStr(EDGE_END1_Y,0) + "]";

		! Calculate and move
		CalcCenterFromEdges;
		DefineWeldLine;

		TPWrite "[MULTI] Calculated R: " + NumToStr(nAngleRzStore,1) + " deg";
		TPWrite "[MULTI] bRobSwap: " + ValToStr(bRobSwap);

		MoveGantryToWeldPosition;

		! Get actual position
		actual_jt := CJointT();
		target_r := actual_jt.extax.eax_d;

		! Calculate TCP tracking
		gantry_physical.x := actual_jt.extax.eax_a;
		gantry_physical.y := actual_jt.extax.eax_b;
		gantry_physical.z := actual_jt.extax.eax_c;
		gantry_floor := PhysicalToFloor(gantry_physical);

		target_floor := calcPosStart;
		offset_floor_x := MODE2_TCP_OFFSET_R1_X * Cos(target_r) - MODE2_TCP_OFFSET_R1_Y * Sin(target_r);
		offset_floor_y := MODE2_TCP_OFFSET_R1_X * Sin(target_r) + MODE2_TCP_OFFSET_R1_Y * Cos(target_r);

		calc_tcp_floor.x := gantry_floor.x + offset_floor_x;
		calc_tcp_floor.y := gantry_floor.y + offset_floor_y;
		calc_tcp_floor.z := gantry_floor.z - WELD_R1_TCP_Z_OFFSET;

		err_x := calc_tcp_floor.x - target_floor.x;
		err_y := calc_tcp_floor.y - target_floor.y;
		err_z := calc_tcp_floor.z - target_floor.z;
		err_total := Sqrt(err_x*err_x + err_y*err_y + err_z*err_z);

		TPWrite "[MULTI] Tracking Error: Total=" + NumToStr(err_total,2) + " mm";

		! Log result
		Write logfile, NumToStr(test_angles{i},0) + " deg | " + NumToStr(test_angles{i},0) + " deg | "
			+ NumToStr(nAngleRzStore,1) + " deg | " + NumToStr(err_x,2) + " | " + NumToStr(err_y,2)
			+ " | " + NumToStr(err_total,2);

		! Wait briefly before next test
		WaitTime 1;
	ENDFOR

	! Restore original edge points
	EDGE_END1_X := orig_end1_x;
	EDGE_END1_Y := orig_end1_y;
	EDGE_END2_X := orig_end2_x;
	EDGE_END2_Y := orig_end2_y;

	! Return to home
	TPWrite "";
	TPWrite "[MULTI] Returning to HOME...";
	ReturnGantryToHome;

	Write logfile, "";
	Write logfile, "Test completed at " + CTime();
	Close logfile;

	TPWrite "";
	TPWrite "========================================";
	TPWrite "[MULTI] Multi-Angle Test Complete";
	TPWrite "[MULTI] Log saved: HOME:/multi_angle_test.txt";
	TPWrite "========================================";
ENDPROC

! ----------------------------------------
! Test Multi-Position: Test various Floor positions (v2.5.0)
! ----------------------------------------
! Tests multiple Floor positions to verify coordinate transformation
! Uses 45deg angle for all tests (consistent with TestMultiAngle)
PROC TestMultiPosition()
	VAR num orig_start1_x;
	VAR num orig_start1_y;
	VAR num orig_start1_z;
	VAR num orig_start2_x;
	VAR num orig_start2_y;
	VAR num orig_start2_z;
	VAR num orig_end1_x;
	VAR num orig_end1_y;
	VAR num orig_end2_x;
	VAR num orig_end2_y;
	VAR num test_x{5};
	VAR num test_y{5};
	VAR num test_z{5};
	VAR string test_name{5};
	VAR num i;
	VAR iodev logfile;
	VAR jointtarget actual_jt;
	VAR pos gantry_physical;
	VAR pos gantry_floor;
	VAR pos target_floor;
	VAR pos calc_tcp_floor;
	VAR num target_r;
	VAR num offset_floor_x;
	VAR num offset_floor_y;
	VAR num err_x;
	VAR num err_y;
	VAR num err_z;
	VAR num err_total;

	TPWrite "========================================";
	TPWrite "[POS] Multi-Position Test v2.5.0";
	TPWrite "========================================";

	! Save original edge points
	orig_start1_x := EDGE_START1_X;
	orig_start1_y := EDGE_START1_Y;
	orig_start1_z := EDGE_START1_Z;
	orig_start2_x := EDGE_START2_X;
	orig_start2_y := EDGE_START2_Y;
	orig_start2_z := EDGE_START2_Z;
	orig_end1_x := EDGE_END1_X;
	orig_end1_y := EDGE_END1_Y;
	orig_end2_x := EDGE_END2_X;
	orig_end2_y := EDGE_END2_Y;

	! Define test positions (Floor coordinates)
	! Position 1: Center (current default)
	test_name{1} := "Center";
	test_x{1} := 5000;
	test_y{1} := 5000;
	test_z{1} := 1200;
	! Position 2: Left side (X smaller)
	test_name{2} := "Left";
	test_x{2} := 3000;
	test_y{2} := 5000;
	test_z{2} := 1200;
	! Position 3: Right side (X larger)
	test_name{3} := "Right";
	test_x{3} := 7000;
	test_y{3} := 5000;
	test_z{3} := 1200;
	! Position 4: Low Z (closer to floor)
	test_name{4} := "LowZ";
	test_x{4} := 5000;
	test_y{4} := 5000;
	test_z{4} := 800;
	! Position 5: High Z (higher up)
	test_name{5} := "HighZ";
	test_x{5} := 5000;
	test_y{5} := 5000;
	test_z{5} := 1600;

	! Open log file
	Open "HOME:/multi_position_test.txt", logfile \Write;
	Write logfile, "Multi-Position Test Log (v2.5.0) - " + CDate() + " " + CTime();
	Write logfile, "";
	Write logfile, "All tests use 45 deg weld line angle";
	Write logfile, "";
	Write logfile, "Position | Floor X,Y,Z | Gantry X,Y,Z,R | Error (mm)";
	Write logfile, "---------+-------------+----------------+-----------";

	! Run tests for each position
	FOR i FROM 1 TO 5 DO
		TPWrite "";
		TPWrite "----------------------------------------";
		TPWrite "[POS] Test " + NumToStr(i,0) + "/5: " + test_name{i};
		TPWrite "[POS] Floor: [" + NumToStr(test_x{i},0) + ", " + NumToStr(test_y{i},0) + ", " + NumToStr(test_z{i},0) + "]";
		TPWrite "----------------------------------------";

		! Set edge points for this position (45deg angle, 500mm weld line)
		! Robot1 side: center Y + 100
		! Robot2 side: center Y - 100
		EDGE_START1_X := test_x{i};
		EDGE_START1_Y := test_y{i} + 100;
		EDGE_START1_Z := test_z{i};
		EDGE_START2_X := test_x{i};
		EDGE_START2_Y := test_y{i} - 100;
		EDGE_START2_Z := test_z{i};
		! End points: 45deg diagonal (dx=354, dy=354)
		EDGE_END1_X := test_x{i} + 354;
		EDGE_END1_Y := test_y{i} + 100 + 354;
		EDGE_END2_X := test_x{i} + 354;
		EDGE_END2_Y := test_y{i} - 100 + 354;

		! Calculate and move
		CalcCenterFromEdges;
		DefineWeldLine;

		TPWrite "[POS] Calculated R: " + NumToStr(nAngleRzStore,1) + " deg";

		MoveGantryToWeldPosition;

		! Get actual position
		actual_jt := CJointT();
		target_r := actual_jt.extax.eax_d;

		! Calculate TCP tracking
		gantry_physical.x := actual_jt.extax.eax_a;
		gantry_physical.y := actual_jt.extax.eax_b;
		gantry_physical.z := actual_jt.extax.eax_c;
		gantry_floor := PhysicalToFloor(gantry_physical);

		target_floor := calcPosStart;
		offset_floor_x := MODE2_TCP_OFFSET_R1_X * Cos(target_r) - MODE2_TCP_OFFSET_R1_Y * Sin(target_r);
		offset_floor_y := MODE2_TCP_OFFSET_R1_X * Sin(target_r) + MODE2_TCP_OFFSET_R1_Y * Cos(target_r);

		calc_tcp_floor.x := gantry_floor.x + offset_floor_x;
		calc_tcp_floor.y := gantry_floor.y + offset_floor_y;
		calc_tcp_floor.z := gantry_floor.z - WELD_R1_TCP_Z_OFFSET;

		err_x := calc_tcp_floor.x - target_floor.x;
		err_y := calc_tcp_floor.y - target_floor.y;
		err_z := calc_tcp_floor.z - target_floor.z;
		err_total := Sqrt(err_x*err_x + err_y*err_y + err_z*err_z);

		TPWrite "[POS] Gantry: X=" + NumToStr(gantry_physical.x,0) + " Y=" + NumToStr(gantry_physical.y,0)
			+ " Z=" + NumToStr(gantry_physical.z,0) + " R=" + NumToStr(target_r,0);
		TPWrite "[POS] Tracking Error: " + NumToStr(err_total,2) + " mm";

		! Log result
		Write logfile, test_name{i} + " | [" + NumToStr(test_x{i},0) + "," + NumToStr(test_y{i},0) + "," + NumToStr(test_z{i},0)
			+ "] | [" + NumToStr(gantry_physical.x,0) + "," + NumToStr(gantry_physical.y,0) + ","
			+ NumToStr(gantry_physical.z,0) + "," + NumToStr(target_r,0) + "] | " + NumToStr(err_total,2);

		! Wait briefly before next test
		WaitTime 1;
	ENDFOR

	! Restore original edge points
	EDGE_START1_X := orig_start1_x;
	EDGE_START1_Y := orig_start1_y;
	EDGE_START1_Z := orig_start1_z;
	EDGE_START2_X := orig_start2_x;
	EDGE_START2_Y := orig_start2_y;
	EDGE_START2_Z := orig_start2_z;
	EDGE_END1_X := orig_end1_x;
	EDGE_END1_Y := orig_end1_y;
	EDGE_END2_X := orig_end2_x;
	EDGE_END2_Y := orig_end2_y;

	! Return to home
	TPWrite "";
	TPWrite "[POS] Returning to HOME...";
	ReturnGantryToHome;

	Write logfile, "";
	Write logfile, "Test completed at " + CTime();
	Close logfile;

	TPWrite "";
	TPWrite "========================================";
	TPWrite "[POS] Multi-Position Test Complete";
	TPWrite "[POS] Log saved: HOME:/multi_position_test.txt";
	TPWrite "========================================";
ENDPROC

! ----------------------------------------
! Move Robot TCP to Weld Position (v2.4.0)
! ----------------------------------------
! Moves Robot1 TCP to the weld start position using WobjGantry
! Call this AFTER gantry is positioned with MoveGantryToWeldPosition
PROC MoveRobotToWeldPosition()
	VAR robtarget weld_target;
	VAR robtarget current_tcp;
	VAR robtarget tcp_floor;
	VAR jointtarget cur_jt;
	VAR jointtarget safe_jt;
	VAR iodev rob_log;

	TPWrite "========================================";
	TPWrite "[ROB] Move Robot to Weld Position v2.5.0";
	TPWrite "========================================";

	! Open log file (overwrite per call - latest move always available)
	Open "HOME:/robot_weld_move.txt", rob_log \Write;
	Write rob_log, "MoveRobotToWeldPosition v2.5.0 - " + CDate() + " " + CTime();
	Write rob_log, "R-axis=" + NumToStr(nAngleRzStore,1) + " bRobSwap=" + ValToStr(bRobSwap);
	Write rob_log, "";

	! Debug: log current joints before any motion
	cur_jt := CJointT();
	Write rob_log, "=== Pre-move (carry-over from previous) ===";
	Write rob_log, "Joints: J1=" + NumToStr(cur_jt.robax.rax_1,1)
		+ " J2=" + NumToStr(cur_jt.robax.rax_2,1)
		+ " J3=" + NumToStr(cur_jt.robax.rax_3,1)
		+ " J4=" + NumToStr(cur_jt.robax.rax_4,1)
		+ " J5=" + NumToStr(cur_jt.robax.rax_5,1)
		+ " J6=" + NumToStr(cur_jt.robax.rax_6,1);
	Write rob_log, "Gantry: X1=" + NumToStr(cur_jt.extax.eax_a,1)
		+ " Y=" + NumToStr(cur_jt.extax.eax_b,1)
		+ " Z=" + NumToStr(cur_jt.extax.eax_c,1)
		+ " R=" + NumToStr(cur_jt.extax.eax_d,1);
	tcp_floor := CRobT(\Tool:=tWeld1\WObj:=WobjFloor);
	Write rob_log, "TCP(Floor): [" + NumToStr(tcp_floor.trans.x,1)
		+ "," + NumToStr(tcp_floor.trans.y,1)
		+ "," + NumToStr(tcp_floor.trans.z,1) + "]";
	TPWrite "[ROB] Pre-move J1=" + NumToStr(cur_jt.robax.rax_1,1)
		+ " J4=" + NumToStr(cur_jt.robax.rax_4,1)
		+ " J5=" + NumToStr(cur_jt.robax.rax_5,1);

	! Step 0: Move robot to safe init joints first (PlanA/PlanC approach)
	! Gantry stays at current position, robot resets to known-good config
	Write rob_log, "";
	Write rob_log, "=== Step 0: Safe init joints ===";
	safe_jt := cur_jt;
	safe_jt.robax.rax_1 := 0;
	safe_jt.robax.rax_2 := -49;
	safe_jt.robax.rax_3 := 6;
	safe_jt.robax.rax_4 := 0;
	safe_jt.robax.rax_5 := 8;
	safe_jt.robax.rax_6 := 0;
	MoveAbsJ safe_jt, v200, fine, tWeld1;

	cur_jt := CJointT();
	Write rob_log, "After safe: J1=" + NumToStr(cur_jt.robax.rax_1,1)
		+ " J2=" + NumToStr(cur_jt.robax.rax_2,1)
		+ " J3=" + NumToStr(cur_jt.robax.rax_3,1)
		+ " J4=" + NumToStr(cur_jt.robax.rax_4,1)
		+ " J5=" + NumToStr(cur_jt.robax.rax_5,1)
		+ " J6=" + NumToStr(cur_jt.robax.rax_6,1);
	tcp_floor := CRobT(\Tool:=tWeld1\WObj:=WobjFloor);
	Write rob_log, "TCP(Floor): [" + NumToStr(tcp_floor.trans.x,1)
		+ "," + NumToStr(tcp_floor.trans.y,1)
		+ "," + NumToStr(tcp_floor.trans.z,1) + "]";
	TPWrite "[ROB] Safe init joints reached";

	! Ensure WobjGantry is updated
	UpdateGantryWobj;

	! Get current TCP position from safe config
	Write rob_log, "";
	Write rob_log, "=== Step 1: Move to weld offset ===";
	current_tcp := CRobT(\Tool:=tWeld1\WObj:=WobjGantry);
	Write rob_log, "Current TCP(WobjGantry): ["
		+ NumToStr(current_tcp.trans.x,1) + ", "
		+ NumToStr(current_tcp.trans.y,1) + ", "
		+ NumToStr(current_tcp.trans.z,1) + "]";
	Write rob_log, "Current orient: ["
		+ NumToStr(current_tcp.rot.q1,5) + ","
		+ NumToStr(current_tcp.rot.q2,5) + ","
		+ NumToStr(current_tcp.rot.q3,5) + ","
		+ NumToStr(current_tcp.rot.q4,5) + "]";
	TPWrite "[ROB] Current TCP (WobjGantry): ["
		+ NumToStr(current_tcp.trans.x,1) + ", "
		+ NumToStr(current_tcp.trans.y,1) + ", "
		+ NumToStr(current_tcp.trans.z,1) + "]";

	! Start with current position (from safe config - predictable robconf/extax/orient)
	weld_target := current_tcp;

	! Define weld target in WobjGantry coordinates
	weld_target.trans.x := 0;
	weld_target.trans.y := MODE2_TCP_OFFSET_R1_Y;

	Write rob_log, "Target TCP(WobjGantry): ["
		+ NumToStr(weld_target.trans.x,1) + ", "
		+ NumToStr(weld_target.trans.y,1) + ", "
		+ NumToStr(weld_target.trans.z,1) + "]";
	Write rob_log, "MODE2_TCP_OFFSET_R1_Y=" + NumToStr(MODE2_TCP_OFFSET_R1_Y,1);
	TPWrite "[ROB] Target TCP (WobjGantry): ["
		+ NumToStr(weld_target.trans.x,1) + ", "
		+ NumToStr(weld_target.trans.y,1) + ", "
		+ NumToStr(weld_target.trans.z,1) + "]";

	! Move robot to weld position (MoveJ from safe config - small, predictable motion)
	TPWrite "[ROB] Moving robot...";
	MoveJ weld_target, v100, fine, tWeld1 \WObj:=WobjGantry;

